KUKA KRL program: EPS_2_25716_MHLP03_A_20250903043914.src

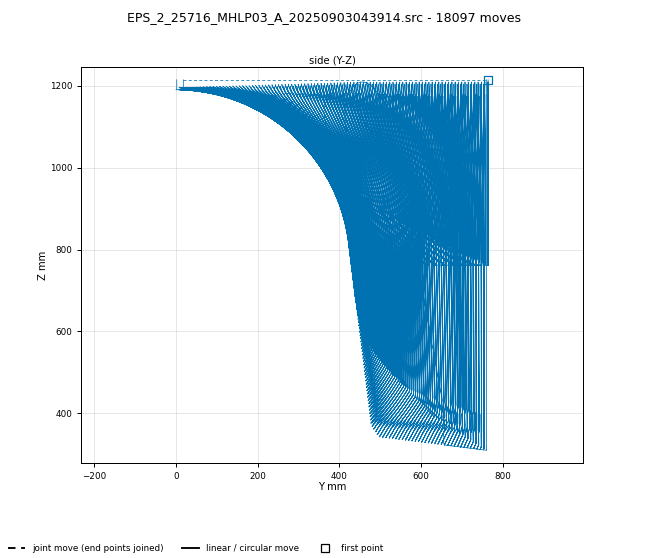
[picture p0: tool path of EPS_2_25716_MHLP03_A_20250903043914.src, 18097 of 18099 moves have a stored position in this frame; points joined in program order, loops and branches not executed]
&ACCESS RVP
&REL 4
&COMMENT QRS 19112012
&PARAM EDITMASK = *
DEF PART()
EXT BAS (BAS_COMMAND :IN,REAL :IN )
INT I
BAS (#INITMOV,0 )

;KUKA QRS Post kuka4.cps  Date:22-06-2017 !

File_ID=2811

QRS_PRE_INIT()

;Init var - Until changes are made in qrs_pre_init
Outlet_Square_prg=0
Inlet_1_Square_prg=0
Inlet_2_Square_prg=0
Inlet_3_Square_prg=0
Inlet_4_Square_prg=0
Inlet_5_Square_prg=0

Outlet_1={X 0.000, Y 457.000, Z 786.000, B 0.000, E1 0.000 }
Inlet_1={X 0.000, Y 514.000, Z 794.000, B 0.000, E1 180.000 }
Outlet_1_type=838
Inlet_1_type=762
;QRS#1=Sidecore dimensions
;QRS#2=825-33" Concrete
;QRS#3=750-30" Concrete
;QRS#4=
;QRS#5=
;QRS#6=
;QRS#7=
;QRS#8=
;QRS#9=S306-46
;QRS#10=S306-42L
;QRS#11=
;QRS#12=
;QRS#13=
;QRS#14=
;QRS#15=
;QRS#16=1524x152x1676 5,5'
;QRS#17=EPS Height
;QRS#18=1205
;QRS#19=*
;QRS#20= UPDATED VERSION 22-06-2017
;QRS#21=*
Outlet_Square=0650
Inlet_1_Square=0550
Inlet_2_Square=0
Inlet_3_Square=0
Inlet_4_Square=0
Inlet_5_Square=0
Mill_Square=1
Outlet_Square_Prg=267
Inlet_1_Square_prg=266

QRS_INIT()

$ADVANCE=5

; T1
PTP {E1 176.609,E2 176.609}
PTP {X 0,Y 763.422,A -85,B 0,C 180,E1 176.609,E2 176.609,E3 0,E4 0,E5 0,E6 0}
QRS_SPEED_INIT()
LIN {X 0,Y 763.422,Z 1215,A -85,B 0,C 180,E1 176.609,E2 176.609,E3 0,E4 0,E5 0,E6 0} C_VEL
LIN {X 0,Y 763.422,Z 764.06,A -85,B 0,C 180,E1 176.609,E2 176.609} C_VEL
LIN {X 0,Y 763.532,Z 762.06,A -85,B 0,C 180,E1 176.759,E2 176.759} C_VEL
LIN {X 0,Y 763.873,Z 762.06,A -85,B 0,C 180,E1 177.187,E2 177.187} C_VEL
LIN {X 0,Y 763.851,Z 762.06,A -85,B 0,C 180,E1 184.692,E2 184.692} C_VEL
LIN {X 0,Y 763.855,Z 762.06,A -85,B 0,C 180,E1 192.28,E2 192.28} C_VEL
LIN {X 0,Y 763.849,Z 762.06,A -85,B 0,C 180,E1 200.095,E2 200.095} C_VEL
LIN {X 0,Y 763.818,Z 762.06,A -85,B 0,C 180,E1 208.325,E2 208.325} C_VEL
LIN {X 0,Y 762.402,Z 762.06,A -85,B 0,C 180,E1 210.54,E2 210.54} C_VEL
LIN {X 0,Y 762.707,Z 762.06,A -85,B 0,C 180,E1 214.993,E2 214.993} C_VEL
LIN {X 0,Y 763.7,Z 762.06,A -85,B 0,C 180,E1 216.696,E2 216.696} C_VEL
LIN {X 0,Y 763.458,Z 762.06,A -85,B 0,C 180,E1 224.738,E2 224.738} C_VEL
LIN {X 0,Y 763.707,Z 762.06,A -85,B 0,C 180,E1 225.281,E2 225.281} C_VEL
LIN {X 0,Y 763.692,Z 762.06,A -85,B 0,C 180,E1 233.306,E2 233.306} C_VEL
LIN {X 0,Y 763.601,Z 762.06,A -85,B 0,C 180,E1 233.585,E2 233.585} C_VEL
LIN {X 0,Y 763.105,Z 765.194,A -85,B 0,C 180,E1 233.692,E2 233.692} C_VEL
LIN {X 0,Y 763.148,Z 825.436,A -85,B 0,C 180,E1 234.391,E2 234.391} C_VEL
LIN {X 0,Y 763.561,Z 841.683,A -85,B 0,C 180,E1 234.66,E2 234.66} C_VEL
LIN {X 0,Y 763.683,Z 859.427,A -85,B 0,C 180,E1 234.998,E2 234.998} C_VEL
LIN {X 0,Y 763.616,Z 876.824,A -85,B 0,C 180,E1 235.383,E2 235.383} C_VEL
LIN {X 0,Y 763.264,Z 892.857,A -85,B 0,C 180,E1 235.785,E2 235.785} C_VEL
LIN {X 0,Y 763.637,Z 914.318,A -85,B 0,C 180,E1 236.454,E2 236.454} C_VEL
LIN {X 0,Y 763.659,Z 936.004,A -85,B 0,C 180,E1 237.219,E2 237.219} C_VEL
LIN {X 0,Y 763.647,Z 955.467,A -85,B 0,C 180,E1 238,E2 238} C_VEL
LIN {X 0,Y 763.481,Z 968.047,A -85,B 0,C 180,E1 238.551,E2 238.551} C_VEL
LIN {X 0,Y 763.561,Z 976.645,A -85,B 0,C 180,E1 238.959,E2 238.959} C_VEL
LIN {X 0,Y 763.516,Z 991.062,A -85,B 0,C 180,E1 239.671,E2 239.671} C_VEL
LIN {X 0,Y 763.481,Z 1008.328,A -85,B 0,C 180,E1 240.608,E2 240.608} C_VEL
LIN {X 0,Y 763.638,Z 1024.577,A -85,B 0,C 180,E1 241.577,E2 241.577} C_VEL
LIN {X 0,Y 763.597,Z 1040.373,A -85,B 0,C 180,E1 242.594,E2 242.594} C_VEL
LIN {X 0,Y 763.3,Z 1055.415,A -85,B 0,C 180,E1 243.634,E2 243.634} C_VEL
LIN {X 0,Y 763.19,Z 1070.039,A -85,B 0,C 180,E1 244.738,E2 244.738} C_VEL
LIN {X 0,Y 763.448,Z 1083.461,A -85,B 0,C 180,E1 245.844,E2 245.844} C_VEL
LIN {X 0,Y 763.685,Z 1096.518,A -85,B 0,C 180,E1 247.003,E2 247.003} C_VEL
LIN {X 0,Y 763.163,Z 1110.025,A -85,B 0,C 180,E1 248.281,E2 248.281} C_VEL
LIN {X 0,Y 762.921,Z 1121.8,A -85,B 0,C 180,E1 249.497,E2 249.497} C_VEL
LIN {X 0,Y 763.255,Z 1133.583,A -85,B 0,C 180,E1 250.839,E2 250.839} C_VEL
LIN {X 0,Y 763.824,Z 1144.005,A -85,B 0,C 180,E1 252.135,E2 252.135} C_VEL
LIN {X 0,Y 763.053,Z 1154.834,A -85,B 0,C 180,E1 253.59,E2 253.59} C_VEL
LIN {X 0,Y 762.741,Z 1164.593,A -85,B 0,C 180,E1 255.058,E2 255.058} C_VEL
LIN {X 0,Y 763.114,Z 1172.36,A -85,B 0,C 180,E1 256.36,E2 256.36} C_VEL
LIN {X 0,Y 763.849,Z 1179.548,A -85,B 0,C 180,E1 257.72,E2 257.72} C_VEL
LIN {X 0,Y 762.886,Z 1187.414,A -85,B 0,C 180,E1 259.38,E2 259.38} C_VEL
LIN {X 0,Y 762.625,Z 1192.231,A -85,B 0,C 180,E1 260.568,E2 260.568} C_VEL
LIN {X 0,Y 762.79,Z 1195.675,A -85,B 0,C 180,E1 261.521,E2 261.521} C_VEL
LIN {X 0,Y 763.28,Z 1198.711,A -85,B 0,C 180,E1 262.474,E2 262.474} C_VEL
LIN {X 0,Y 763.858,Z 1201.343,A -85,B 0,C 180,E1 263.424,E2 263.424} C_VEL
LIN {X 0,Y 763.266,Z 1203.657,A -85,B 0,C 180,E1 264.362,E2 264.362} C_VEL
LIN {X 0,Y 762.79,Z 1205.612,A -85,B 0,C 180,E1 265.301,E2 265.301} C_VEL
LIN {X 0,Y 762.61,Z 1207.201,A -85,B 0,C 180,E1 266.242,E2 266.242} C_VEL
LIN {X 0,Y 762.976,Z 1208.861,A -85,B 0,C 180,E1 267.626,E2 267.626} C_VEL
LIN {X 0,Y 763.872,Z 1209.666,A -85,B 0,C 180,E1 269.062,E2 269.062} C_VEL
LIN {X 0,Y 762.824,Z 1209.715,A -85,B 0,C 180,E1 270.939,E2 270.939} C_VEL
LIN {X 0,Y 762.627,Z 1209.463,A -85,B 0,C 180,E1 271.621,E2 271.621} C_VEL
LIN {X 0,Y 762.799,Z 1208.402,A -85,B 0,C 180,E1 272.817,E2 272.817} C_VEL
LIN {X 0,Y 763.272,Z 1207.185,A -85,B 0,C 180,E1 273.755,E2 273.755} C_VEL
LIN {X 0,Y 763.867,Z 1205.576,A -85,B 0,C 180,E1 274.692,E2 274.692} C_VEL
LIN {X 0,Y 763.013,Z 1202.588,A -85,B 0,C 180,E1 276.111,E2 276.111} C_VEL
LIN {X 0,Y 762.637,Z 1198.716,A -85,B 0,C 180,E1 277.533,E2 277.533} C_VEL
LIN {X 0,Y 762.799,Z 1195.676,A -85,B 0,C 180,E1 278.479,E2 278.479} C_VEL
LIN {X 0,Y 763.569,Z 1190.398,A -85,B 0,C 180,E1 279.895,E2 279.895} C_VEL
LIN {X 0,Y 763.864,Z 1188.41,A -85,B 0,C 180,E1 280.367,E2 280.367} C_VEL
LIN {X 0,Y 763.206,Z 1182.983,A -85,B 0,C 180,E1 281.571,E2 281.571} C_VEL
LIN {X 0,Y 762.859,Z 1179.549,A -85,B 0,C 180,E1 282.296,E2 282.296} C_VEL
LIN {X 0,Y 762.736,Z 1172.081,A -85,B 0,C 180,E1 283.695,E2 283.695} C_VEL
LIN {X 0,Y 763.29,Z 1163.915,A -85,B 0,C 180,E1 285.044,E2 285.044} C_VEL
LIN {X 0,Y 763.763,Z 1158.34,A -85,B 0,C 180,E1 285.871,E2 285.871} C_VEL
LIN {X 0,Y 763.637,Z 1154.836,A -85,B 0,C 180,E1 286.397,E2 286.397} C_VEL
LIN {X 0,Y 762.912,Z 1144.007,A -85,B 0,C 180,E1 287.886,E2 287.886} C_VEL
LIN {X 0,Y 762.868,Z 1132,A -85,B 0,C 180,E1 289.358,E2 289.358} C_VEL
LIN {X 0,Y 763.42,Z 1120.423,A -85,B 0,C 180,E1 290.638,E2 290.638} C_VEL
LIN {X 0,Y 763.768,Z 1112.185,A -85,B 0,C 180,E1 291.477,E2 291.477} C_VEL
LIN {X 0,Y 763.558,Z 1105.856,A -85,B 0,C 180,E1 292.113,E2 292.113} C_VEL
LIN {X 0,Y 763.217,Z 1095.11,A -85,B 0,C 180,E1 293.14,E2 293.14} C_VEL
LIN {X 0,Y 763.154,Z 1081.968,A -85,B 0,C 180,E1 294.292,E2 294.292} C_VEL
LIN {X 0,Y 763.464,Z 1068.228,A -85,B 0,C 180,E1 295.394,E2 295.394} C_VEL
LIN {X 0,Y 763.662,Z 1053.606,A -85,B 0,C 180,E1 296.483,E2 296.483} C_VEL
LIN {X 0,Y 763.467,Z 1037.367,A -85,B 0,C 180,E1 297.609,E2 297.609} C_VEL
LIN {X 0,Y 763.402,Z 1021.787,A -85,B 0,C 180,E1 298.602,E2 298.602} C_VEL
LIN {X 0,Y 763.565,Z 1005.34,A -85,B 0,C 180,E1 299.557,E2 299.557} C_VEL
LIN {X 0,Y 763.602,Z 989.459,A -85,B 0,C 180,E1 300.411,E2 300.411} C_VEL
LIN {X 0,Y 763.621,Z 970.475,A -85,B 0,C 180,E1 301.335,E2 301.335} C_VEL
LIN {X 0,Y 763.591,Z 951.701,A -85,B 0,C 180,E1 302.16,E2 302.16} C_VEL
LIN {X 0,Y 763.574,Z 933.239,A -85,B 0,C 180,E1 302.888,E2 302.888} C_VEL
LIN {X 0,Y 763.35,Z 920.5,A -85,B 0,C 180,E1 303.348,E2 303.348} C_VEL
LIN {X 0,Y 763.571,Z 911.932,A -85,B 0,C 180,E1 303.623,E2 303.623} C_VEL
LIN {X 0,Y 763.721,Z 893.145,A -85,B 0,C 180,E1 304.183,E2 304.183} C_VEL
LIN {X 0,Y 763.708,Z 876.573,A -85,B 0,C 180,E1 304.618,E2 304.618} C_VEL
LIN {X 0,Y 763.517,Z 859.345,A -85,B 0,C 180,E1 305.013,E2 305.013} C_VEL
LIN {X 0,Y 763.205,Z 848.039,A -85,B 0,C 180,E1 305.249,E2 305.249} C_VEL
LIN {X 0,Y 763.489,Z 831.099,A -85,B 0,C 180,E1 305.51,E2 305.51} C_VEL
LIN {X 0,Y 763.501,Z 819.142,A -85,B 0,C 180,E1 305.669,E2 305.669} C_VEL
LIN {X 0,Y 763.102,Z 762.521,A -85,B 0,C 180,E1 306.339,E2 306.339} C_VEL
LIN {X 0,Y 763.722,Z 762.06,A -85,B 0,C 180,E1 306.444,E2 306.444} C_VEL
LIN {X 0,Y 763.585,Z 762.06,A -85,B 0,C 180,E1 306.961,E2 306.961} C_VEL
LIN {X 0,Y 763.809,Z 762.06,A -85,B 0,C 180,E1 312.129,E2 312.129} C_VEL
LIN {X 0,Y 763.614,Z 762.06,A -85,B 0,C 180,E1 312.57,E2 312.57} C_VEL
LIN {X 0,Y 763.761,Z 762.06,A -85,B 0,C 180,E1 320.266,E2 320.266} C_VEL
LIN {X 0,Y 763.673,Z 762.06,A -85,B 0,C 180,E1 326.571,E2 326.571} C_VEL
LIN {X 0,Y 763.435,Z 762.06,A -85,B 0,C 180,E1 327.303,E2 327.303} C_VEL
LIN {X 0,Y 763.817,Z 762.06,A -85,B 0,C 180,E1 333.784,E2 333.784} C_VEL
LIN {X 0,Y 763.847,Z 762.06,A -85,B 0,C 180,E1 341.889,E2 341.889} C_VEL
LIN {X 0,Y 763.863,Z 762.06,A -85,B 0,C 180,E1 349.632,E2 349.632} C_VEL
LIN {X 0,Y 763.842,Z 762.06,A -85,B 0,C 180,E1 357.187,E2 357.187} C_VEL
LIN {X 0,Y 763.858,Z 762.06,A -85,B 0,C 180,E1 364.692,E2 364.692} C_VEL
LIN {X 0,Y 763.826,Z 762.06,A -85,B 0,C 180,E1 372.28,E2 372.28} C_VEL
LIN {X 0,Y 763.82,Z 762.06,A -85,B 0,C 180,E1 380.096,E2 380.096} C_VEL
LIN {X 0,Y 763.775,Z 762.06,A -85,B 0,C 180,E1 388.327,E2 388.327} C_VEL
LIN {X 0,Y 763.769,Z 762.06,A -85,B 0,C 180,E1 394.938,E2 394.938} C_VEL
LIN {X 0,Y 762.467,Z 762.06,A -85,B 0,C 180,E1 399.734,E2 399.734} C_VEL
LIN {X 0,Y 763.757,Z 762.06,A -85,B 0,C 180,E1 402.134,E2 402.134} C_VEL
LIN {X 0,Y 763.589,Z 762.06,A -85,B 0,C 180,E1 402.569,E2 402.569} C_VEL
LIN {X 0,Y 763.857,Z 762.06,A -85,B 0,C 180,E1 410.259,E2 410.259} C_VEL
LIN {X 0,Y 763.738,Z 762.06,A -85,B 0,C 180,E1 416.565,E2 416.565} C_VEL
LIN {X 0,Y 763.397,Z 762.06,A -85,B 0,C 180,E1 416.915,E2 416.915} C_VEL
LIN {X 0,Y 762.602,Z 762.061,A -85,B 0,C 180,E1 416.991,E2 416.991} C_VEL
LIN {X 0,Y 763.35,Z 823.326,A -85,B 0,C 180,E1 417.706,E2 417.706} C_VEL
LIN {X 0,Y 763.333,Z 838.865,A -85,B 0,C 180,E1 417.911,E2 417.911} C_VEL
LIN {X 0,Y 763.673,Z 858.064,A -85,B 0,C 180,E1 418.263,E2 418.263} C_VEL
LIN {X 0,Y 763.723,Z 875.941,A -85,B 0,C 180,E1 418.651,E2 418.651} C_VEL
LIN {X 0,Y 763.595,Z 893.845,A -85,B 0,C 180,E1 419.106,E2 419.106} C_VEL
LIN {X 0,Y 763.455,Z 902.424,A -85,B 0,C 180,E1 419.354,E2 419.354} C_VEL
LIN {X 0,Y 763.674,Z 913.5,A -85,B 0,C 180,E1 419.706,E2 419.706} C_VEL
LIN {X 0,Y 763.678,Z 930.085,A -85,B 0,C 180,E1 420.28,E2 420.28} C_VEL
LIN {X 0,Y 763.697,Z 947.445,A -85,B 0,C 180,E1 420.959,E2 420.959} C_VEL
LIN {X 0,Y 763.678,Z 963.783,A -85,B 0,C 180,E1 421.67,E2 421.67} C_VEL
LIN {X 0,Y 763.609,Z 974.911,A -85,B 0,C 180,E1 422.198,E2 422.198} C_VEL
LIN {X 0,Y 763.613,Z 984.032,A -85,B 0,C 180,E1 422.661,E2 422.661} C_VEL
LIN {X 0,Y 763.513,Z 996.348,A -85,B 0,C 180,E1 423.315,E2 423.315} C_VEL
LIN {X 0,Y 763.537,Z 1011.273,A -85,B 0,C 180,E1 424.185,E2 424.185} C_VEL
LIN {X 0,Y 763.684,Z 1026.123,A -85,B 0,C 180,E1 425.134,E2 425.134} C_VEL
LIN {X 0,Y 763.619,Z 1038.484,A -85,B 0,C 180,E1 425.978,E2 425.978} C_VEL
LIN {X 0,Y 763.318,Z 1052.22,A -85,B 0,C 180,E1 426.991,E2 426.991} C_VEL
LIN {X 0,Y 763.258,Z 1064.783,A -85,B 0,C 180,E1 428.003,E2 428.003} C_VEL
LIN {X 0,Y 763.568,Z 1077.587,A -85,B 0,C 180,E1 429.134,E2 429.134} C_VEL
LIN {X 0,Y 763.744,Z 1087.004,A -85,B 0,C 180,E1 430.024,E2 430.024} C_VEL
LIN {X 0,Y 763.2,Z 1099.807,A -85,B 0,C 180,E1 431.321,E2 431.321} C_VEL
LIN {X 0,Y 763.019,Z 1110.232,A -85,B 0,C 180,E1 432.486,E2 432.486} C_VEL
LIN {X 0,Y 763.299,Z 1119.275,A -85,B 0,C 180,E1 433.595,E2 433.595} C_VEL
LIN {X 0,Y 763.838,Z 1128.649,A -85,B 0,C 180,E1 434.861,E2 434.861} C_VEL
LIN {X 0,Y 763.059,Z 1138.172,A -85,B 0,C 180,E1 436.263,E2 436.263} C_VEL
LIN {X 0,Y 762.712,Z 1144.936,A -85,B 0,C 180,E1 437.381,E2 437.381} C_VEL
LIN {X 0,Y 763.034,Z 1153.093,A -85,B 0,C 180,E1 438.905,E2 438.905} C_VEL
LIN {X 0,Y 763.728,Z 1158.659,A -85,B 0,C 180,E1 440.107,E2 440.107} C_VEL
LIN {X 0,Y 763.702,Z 1160.649,A -85,B 0,C 180,E1 440.582,E2 440.582} C_VEL
LIN {X 0,Y 763.147,Z 1164.462,A -85,B 0,C 180,E1 441.525,E2 441.525} C_VEL
LIN {X 0,Y 762.699,Z 1169.301,A -85,B 0,C 180,E1 442.941,E2 442.941} C_VEL
LIN {X 0,Y 763.043,Z 1173.205,A -85,B 0,C 180,E1 444.361,E2 444.361} C_VEL
LIN {X 0,Y 763.604,Z 1175.195,A -85,B 0,C 180,E1 445.306,E2 445.306} C_VEL
LIN {X 0,Y 763.572,Z 1176.903,A -85,B 0,C 180,E1 446.247,E2 446.247} C_VEL
LIN {X 0,Y 762.964,Z 1178.329,A -85,B 0,C 180,E1 447.184,E2 447.184} C_VEL
LIN {X 0,Y 762.58,Z 1179.53,A -85,B 0,C 180,E1 448.508,E2 448.508} C_VEL
LIN {X 0,Y 762.643,Z 1179.734,A -85,B 0,C 180,E1 449.061,E2 449.061} C_VEL
LIN {X 0,Y 763.561,Z 1179.673,A -85,B 0,C 180,E1 450.938,E2 450.938} C_VEL
LIN {X 0,Y 763.13,Z 1178.412,A -85,B 0,C 180,E1 452.638,E2 452.638} C_VEL
LIN {X 0,Y 762.743,Z 1176.796,A -85,B 0,C 180,E1 453.758,E2 453.758} C_VEL
LIN {X 0,Y 762.944,Z 1174.031,A -85,B 0,C 180,E1 455.169,E2 455.169} C_VEL
LIN {X 0,Y 763.153,Z 1172.957,A -85,B 0,C 180,E1 455.639,E2 455.639} C_VEL
LIN {X 0,Y 763.71,Z 1170.361,A -85,B 0,C 180,E1 456.577,E2 456.577} C_VEL
LIN {X 0,Y 763.728,Z 1168.983,A -85,B 0,C 180,E1 457.049,E2 457.049} C_VEL
LIN {X 0,Y 762.942,Z 1164.1,A -85,B 0,C 180,E1 458.477,E2 458.477} C_VEL
LIN {X 0,Y 762.689,Z 1159.333,A -85,B 0,C 180,E1 459.669,E2 459.669} C_VEL
LIN {X 0,Y 763.153,Z 1152.641,A -85,B 0,C 180,E1 461.094,E2 461.094} C_VEL
LIN {X 0,Y 763.854,Z 1146.251,A -85,B 0,C 180,E1 462.28,E2 462.28} C_VEL
LIN {X 0,Y 763.151,Z 1138.199,A -85,B 0,C 180,E1 463.641,E2 463.641} C_VEL
LIN {X 0,Y 762.78,Z 1128.325,A -85,B 0,C 180,E1 465.114,E2 465.114} C_VEL
LIN {X 0,Y 763.189,Z 1118.534,A -85,B 0,C 180,E1 466.407,E2 466.407} C_VEL
LIN {X 0,Y 763.808,Z 1108.38,A -85,B 0,C 180,E1 467.619,E2 467.619} C_VEL
LIN {X 0,Y 763.383,Z 1098.021,A -85,B 0,C 180,E1 468.775,E2 468.775} C_VEL
LIN {X 0,Y 763.102,Z 1086.005,A -85,B 0,C 180,E1 469.997,E2 469.997} C_VEL
LIN {X 0,Y 763.291,Z 1074.606,A -85,B 0,C 180,E1 471.054,E2 471.054} C_VEL
LIN {X 0,Y 763.698,Z 1062.183,A -85,B 0,C 180,E1 472.109,E2 472.109} C_VEL
LIN {X 0,Y 763.642,Z 1051.08,A -85,B 0,C 180,E1 472.999,E2 472.999} C_VEL
LIN {X 0,Y 763.363,Z 1037.208,A -85,B 0,C 180,E1 474.031,E2 474.031} C_VEL
LIN {X 0,Y 763.39,Z 1022.484,A -85,B 0,C 180,E1 475.026,E2 475.026} C_VEL
LIN {X 0,Y 763.608,Z 1007.982,A -85,B 0,C 180,E1 475.922,E2 475.922} C_VEL
LIN {X 0,Y 763.681,Z 992.341,A -85,B 0,C 180,E1 476.81,E2 476.81} C_VEL
LIN {X 0,Y 763.637,Z 977.185,A -85,B 0,C 180,E1 477.602,E2 477.602} C_VEL
LIN {X 0,Y 763.612,Z 960.801,A -85,B 0,C 180,E1 478.379,E2 478.379} C_VEL
LIN {X 0,Y 763.629,Z 942.917,A -85,B 0,C 180,E1 479.138,E2 479.138} C_VEL
LIN {X 0,Y 763.481,Z 932.728,A -85,B 0,C 180,E1 479.536,E2 479.536} C_VEL
LIN {X 0,Y 763.665,Z 923.871,A -85,B 0,C 180,E1 479.851,E2 479.851} C_VEL
LIN {X 0,Y 763.752,Z 908.211,A -85,B 0,C 180,E1 480.371,E2 480.371} C_VEL
LIN {X 0,Y 763.742,Z 891.43,A -85,B 0,C 180,E1 480.865,E2 480.865} C_VEL
LIN {X 0,Y 763.585,Z 872.972,A -85,B 0,C 180,E1 481.335,E2 481.335} C_VEL
LIN {X 0,Y 763.349,Z 865.666,A -85,B 0,C 180,E1 481.501,E2 481.501} C_VEL
LIN {X 0,Y 763.643,Z 854.355,A -85,B 0,C 180,E1 481.72,E2 481.72} C_VEL
LIN {X 0,Y 763.767,Z 835.648,A -85,B 0,C 180,E1 482.025,E2 482.025} C_VEL
LIN {X 0,Y 763.645,Z 814.716,A -85,B 0,C 180,E1 482.292,E2 482.292} C_VEL
LIN {X 0,Y 763.119,Z 784.369,A -85,B 0,C 180,E1 482.649,E2 482.649} C_VEL
LIN {X 0,Y 761.841,Z 762.933,A -85,B 0,C 180,E1 482.946,E2 482.946} C_VEL
LIN {X 0,Y 761.836,Z 762.06,A -85,B 0,C 180,E1 482.963,E2 482.963} C_VEL
LIN {X 0,Y 762.124,Z 762.06,A -85,B 0,C 180,E1 482.976,E2 482.976} C_VEL
LIN {X 0,Y 763.606,Z 762.06,A -85,B 0,C 180,E1 483.119,E2 483.119} C_VEL
LIN {X 0,Y 763.812,Z 762.06,A -85,B 0,C 180,E1 483.443,E2 483.443} C_VEL
LIN {X 0,Y 763.69,Z 762.06,A -85,B 0,C 180,E1 486.694,E2 486.694} C_VEL
LIN {X 0,Y 763.69,Z 762.06,A -85,B 0,C 180,E1 494.72,E2 494.72} C_VEL
LIN {X 0,Y 763.483,Z 762.06,A -85,B 0,C 180,E1 495.264,E2 495.264} C_VEL
LIN {X 0,Y 762.408,Z 762.06,A -85,B 0,C 180,E1 500.389,E2 500.389} C_VEL
LIN {X 0,Y 763.783,Z 762.06,A -85,B 0,C 180,E1 502.743,E2 502.743} C_VEL
LIN {X 0,Y 763.683,Z 762.06,A -85,B 0,C 180,E1 510.145,E2 510.145} C_VEL
LIN {X 0,Y 762.968,Z 762.06,A -85,B 0,C 180,E1 511.64,E2 511.64} C_VEL
LIN {X 0,Y 763.8,Z 762.06,A -85,B 0,C 180,E1 517.894,E2 517.894} C_VEL
LIN {X 0,Y 763.495,Z 762.06,A -85,B 0,C 180,E1 524.953,E2 524.953} C_VEL
LIN {X 0,Y 763.693,Z 762.06,A -85,B 0,C 180,E1 525.791,E2 525.791} C_VEL
LIN {X 0,Y 763.845,Z 762.06,A -85,B 0,C 180,E1 529.632,E2 529.632} C_VEL
LIN {X 0,Y 763.532,Z 762.06,A -85,B 0,C 180,E1 536.759,E2 536.759} C_VEL
LIN {X 0,Y 754.518,Z 762.06,A -85,B 0,C 180,E1 539.358,E2 539.358} C_VEL
LIN {X 0,Y 754.715,Z 762.06,A -85,B 0,C 180,E1 546.362,E2 546.362} C_VEL
LIN {X 0,Y 755.003,Z 762.06,A -85,B 0,C 180,E1 553.379,E2 553.379} C_VEL
LIN {X 0,Y 755.112,Z 762.06,A -85,B 0,C 180,E1 560.95,E2 560.95} C_VEL
LIN {X 0,Y 754.911,Z 762.06,A -85,B 0,C 180,E1 569.525,E2 569.525} C_VEL
LIN {X 0,Y 754.735,Z 762.06,A -85,B 0,C 180,E1 577.848,E2 577.848} C_VEL
LIN {X 0,Y 754.995,Z 762.06,A -85,B 0,C 180,E1 586.132,E2 586.132} C_VEL
LIN {X 0,Y 755.889,Z 764.005,A -85,B 0,C 180,E1 593.275,E2 593.275} C_VEL
LIN {X 0,Y 757.067,Z 866.417,A -85,B 0,C 180,E1 594.797,E2 594.797} C_VEL
LIN {X 0,Y 756.732,Z 937.533,A -85,B 0,C 180,E1 596.942,E2 596.942} C_VEL
LIN {X 0,Y 756.224,Z 1008.772,A -85,B 0,C 180,E1 600.324,E2 600.324} C_VEL
LIN {X 0,Y 755.596,Z 1073.515,A -85,B 0,C 180,E1 604.753,E2 604.753} C_VEL
LIN {X 0,Y 755.135,Z 1125.789,A -85,B 0,C 180,E1 609.73,E2 609.73} C_VEL
LIN {X 0,Y 754.862,Z 1162.477,A -85,B 0,C 180,E1 614.561,E2 614.561} C_VEL
LIN {X 0,Y 754.828,Z 1188.719,A -85,B 0,C 180,E1 619.581,E2 619.581} C_VEL
LIN {X 0,Y 755.026,Z 1204.76,A -85,B 0,C 180,E1 624.813,E2 624.813} C_VEL
LIN {X 0,Y 755.621,Z 1209.837,A -85,B 0,C 180,E1 629.424,E2 629.424} C_VEL
LIN {X 0,Y 755.519,Z 1204.764,A -85,B 0,C 180,E1 635.181,E2 635.181} C_VEL
LIN {X 0,Y 755.373,Z 1184.858,A -85,B 0,C 180,E1 641.287,E2 641.287} C_VEL
LIN {X 0,Y 755.345,Z 1150.798,A -85,B 0,C 180,E1 647.144,E2 647.144} C_VEL
LIN {X 0,Y 755.668,Z 1103.645,A -85,B 0,C 180,E1 652.569,E2 652.569} C_VEL
LIN {X 0,Y 756.059,Z 1043.633,A -85,B 0,C 180,E1 657.472,E2 657.472} C_VEL
LIN {X 0,Y 756.496,Z 976.301,A -85,B 0,C 180,E1 661.381,E2 661.381} C_VEL
LIN {X 0,Y 756.901,Z 903.888,A -85,B 0,C 180,E1 664.21,E2 664.21} C_VEL
LIN {X 0,Y 756.982,Z 829.369,A -85,B 0,C 180,E1 665.888,E2 665.888} C_VEL
LIN {X 0,Y 755.632,Z 762.06,A -85,B 0,C 180,E1 666.796,E2 666.796} C_VEL
LIN {X 0,Y 754.653,Z 762.06,A -85,B 0,C 180,E1 673.89,E2 673.89} C_VEL
LIN {X 0,Y 754.78,Z 762.06,A -85,B 0,C 180,E1 682.154,E2 682.154} C_VEL
LIN {X 0,Y 754.74,Z 762.06,A -85,B 0,C 180,E1 688.643,E2 688.643} C_VEL
LIN {X 0,Y 755.303,Z 762.06,A -85,B 0,C 180,E1 694.389,E2 694.389} C_VEL
LIN {X 0,Y 754.964,Z 762.06,A -85,B 0,C 180,E1 703.039,E2 703.039} C_VEL
LIN {X 0,Y 755.425,Z 762.06,A -85,B 0,C 180,E1 710.155,E2 710.155} C_VEL
LIN {X 0,Y 755.038,Z 762.06,A -85,B 0,C 180,E1 718.26,E2 718.26} C_VEL
LIN {X 0,Y 754.869,Z 762.06,A -85,B 0,C 180,E1 726.055,E2 726.055} C_VEL
LIN {X 0,Y 754.978,Z 762.06,A -85,B 0,C 180,E1 733.355,E2 733.355} C_VEL
LIN {X 0,Y 755.074,Z 762.06,A -85,B 0,C 180,E1 740.949,E2 740.949} C_VEL
LIN {X 0,Y 755.031,Z 762.06,A -85,B 0,C 180,E1 749.492,E2 749.492} C_VEL
LIN {X 0,Y 754.827,Z 762.06,A -85,B 0,C 180,E1 756.369,E2 756.369} C_VEL
LIN {X 0,Y 755.347,Z 762.06,A -85,B 0,C 180,E1 762.879,E2 762.879} C_VEL
LIN {X 0,Y 755.489,Z 762.06,A -85,B 0,C 180,E1 770.781,E2 770.781} C_VEL
LIN {X 0,Y 755.761,Z 763.481,A -85,B 0,C 180,E1 776.67,E2 776.67} C_VEL
LIN {X 0,Y 756.835,Z 867.232,A -85,B 0,C 180,E1 778.14,E2 778.14} C_VEL
LIN {X 0,Y 756.556,Z 937.416,A -85,B 0,C 180,E1 780.258,E2 780.258} C_VEL
LIN {X 0,Y 756.087,Z 1005.684,A -85,B 0,C 180,E1 783.576,E2 783.576} C_VEL
LIN {X 0,Y 755.561,Z 1064.464,A -85,B 0,C 180,E1 787.739,E2 787.739} C_VEL
LIN {X 0,Y 755.151,Z 1110.654,A -85,B 0,C 180,E1 792.35,E2 792.35} C_VEL
LIN {X 0,Y 754.843,Z 1143.269,A -85,B 0,C 180,E1 796.968,E2 796.968} C_VEL
LIN {X 0,Y 754.988,Z 1166.131,A -85,B 0,C 180,E1 801.918,E2 801.918} C_VEL
LIN {X 0,Y 755.023,Z 1178.299,A -85,B 0,C 180,E1 807.123,E2 807.123} C_VEL
LIN {X 0,Y 755.288,Z 1179.26,A -85,B 0,C 180,E1 811.727,E2 811.727} C_VEL
LIN {X 0,Y 755.439,Z 1167.758,A -85,B 0,C 180,E1 817.499,E2 817.499} C_VEL
LIN {X 0,Y 755.48,Z 1142.577,A -85,B 0,C 180,E1 823.047,E2 823.047} C_VEL
LIN {X 0,Y 755.644,Z 1102.95,A -85,B 0,C 180,E1 828.428,E2 828.428} C_VEL
LIN {X 0,Y 755.962,Z 1050.543,A -85,B 0,C 180,E1 833.287,E2 833.287} C_VEL
LIN {X 0,Y 756.297,Z 988.391,A -85,B 0,C 180,E1 837.304,E2 837.304} C_VEL
LIN {X 0,Y 756.657,Z 919.117,A -85,B 0,C 180,E1 840.32,E2 840.32} C_VEL
LIN {X 0,Y 756.897,Z 847.457,A -85,B 0,C 180,E1 842.156,E2 842.156} C_VEL
LIN {X 0,Y 755.541,Z 762.06,A -85,B 0,C 180,E1 843.332,E2 843.332} C_VEL
LIN {X 0,Y 754.065,Z 762.06,A -85,B 0,C 180,E1 849.31,E2 849.31} C_VEL
LIN {X 0,Y 754.889,Z 762.06,A -85,B 0,C 180,E1 856.095,E2 856.095} C_VEL
LIN {X 0,Y 755.09,Z 762.06,A -85,B 0,C 180,E1 863.646,E2 863.646} C_VEL
LIN {X 0,Y 754.879,Z 762.06,A -85,B 0,C 180,E1 871.816,E2 871.816} C_VEL
LIN {X 0,Y 754.77,Z 762.06,A -85,B 0,C 180,E1 879.408,E2 879.408} C_VEL
LIN {X 0,Y 755.411,Z 762.06,A -85,B 0,C 180,E1 886.824,E2 886.824} C_VEL
LIN {X 0,Y 754.221,Z 762.06,A -85,B 0,C 180,E1 893.657,E2 893.657} C_VEL
LIN {X 0,Y 755.069,Z 762.06,A -85,B 0,C 180,E1 898.284,E2 898.284} C_VEL
LIN {X 0,Y 754.518,Z 762.06,A -85,B 0,C 180,E1 899.358,E2 899.358} C_VEL
LIN {X 0,Y 746.381,Z 762.06,A -85,B 0,C 180,E1 901.989,E2 901.989} C_VEL
LIN {X 0,Y 746.269,Z 762.06,A -85,B 0,C 180,E1 907.609,E2 907.609} C_VEL
LIN {X 0,Y 746.903,Z 762.06,A -85,B 0,C 180,E1 913.527,E2 913.527} C_VEL
LIN {X 0,Y 747.198,Z 762.06,A -85,B 0,C 180,E1 920.836,E2 920.836} C_VEL
LIN {X 0,Y 747.486,Z 762.06,A -85,B 0,C 180,E1 928.515,E2 928.515} C_VEL
LIN {X 0,Y 747.242,Z 762.06,A -85,B 0,C 180,E1 936.828,E2 936.828} C_VEL
LIN {X 0,Y 746.946,Z 762.06,A -85,B 0,C 180,E1 946.184,E2 946.184} C_VEL
LIN {X 0,Y 747.356,Z 763.412,A -85,B 0,C 180,E1 952.778,E2 952.778} C_VEL
LIN {X 0,Y 750.226,Z 775.649,A -85,B 0,C 180,E1 953.088,E2 953.088} C_VEL
LIN {X 0,Y 750.485,Z 865.241,A -85,B 0,C 180,E1 954.415,E2 954.415} C_VEL
LIN {X 0,Y 749.898,Z 935.677,A -85,B 0,C 180,E1 956.526,E2 956.526} C_VEL
LIN {X 0,Y 749.014,Z 1006.369,A -85,B 0,C 180,E1 959.866,E2 959.866} C_VEL
LIN {X 0,Y 748.042,Z 1071.316,A -85,B 0,C 180,E1 964.296,E2 964.296} C_VEL
LIN {X 0,Y 747.318,Z 1123.096,A -85,B 0,C 180,E1 969.198,E2 969.198} C_VEL
LIN {X 0,Y 747.022,Z 1160.497,A -85,B 0,C 180,E1 974.093,E2 974.093} C_VEL
LIN {X 0,Y 747,Z 1187.51,A -85,B 0,C 180,E1 979.175,E2 979.175} C_VEL
LIN {X 0,Y 747.062,Z 1204.76,A -85,B 0,C 180,E1 984.758,E2 984.758} C_VEL
LIN {X 0,Y 747.615,Z 1209.837,A -85,B 0,C 180,E1 989.418,E2 989.418} C_VEL
LIN {X 0,Y 747.495,Z 1204.764,A -85,B 0,C 180,E1 995.237,E2 995.237} C_VEL
LIN {X 0,Y 747.349,Z 1184.859,A -85,B 0,C 180,E1 1001.41,E2 1001.41} C_VEL
LIN {X 0,Y 747.385,Z 1151.064,A -85,B 0,C 180,E1 1007.296,E2 1007.296} C_VEL
LIN {X 0,Y 747.909,Z 1103.128,A -85,B 0,C 180,E1 1012.866,E2 1012.866} C_VEL
LIN {X 0,Y 748.596,Z 1043.549,A -85,B 0,C 180,E1 1017.776,E2 1017.776} C_VEL
LIN {X 0,Y 749.437,Z 974.405,A -85,B 0,C 180,E1 1021.807,E2 1021.807} C_VEL
LIN {X 0,Y 750.191,Z 902.761,A -85,B 0,C 180,E1 1024.595,E2 1024.595} C_VEL
LIN {X 0,Y 750.507,Z 828.895,A -85,B 0,C 180,E1 1026.253,E2 1026.253} C_VEL
LIN {X 0,Y 748.657,Z 766.226,A -85,B 0,C 180,E1 1027.113,E2 1027.113} C_VEL
LIN {X 0,Y 747.392,Z 762.06,A -85,B 0,C 180,E1 1027.323,E2 1027.323} C_VEL
LIN {X 0,Y 746.72,Z 762.06,A -85,B 0,C 180,E1 1033.797,E2 1033.797} C_VEL
LIN {X 0,Y 746.941,Z 762.06,A -85,B 0,C 180,E1 1041.686,E2 1041.686} C_VEL
LIN {X 0,Y 746.71,Z 762.06,A -85,B 0,C 180,E1 1048.766,E2 1048.766} C_VEL
LIN {X 0,Y 746.635,Z 762.06,A -85,B 0,C 180,E1 1055.358,E2 1055.358} C_VEL
LIN {X 0,Y 747.083,Z 762.06,A -85,B 0,C 180,E1 1062.855,E2 1062.855} C_VEL
LIN {X 0,Y 746.761,Z 762.06,A -85,B 0,C 180,E1 1071.22,E2 1071.22} C_VEL
LIN {X 0,Y 747.042,Z 762.06,A -85,B 0,C 180,E1 1078.242,E2 1078.242} C_VEL
LIN {X 0,Y 747.42,Z 762.06,A -85,B 0,C 180,E1 1085.231,E2 1085.231} C_VEL
LIN {X 0,Y 746.878,Z 762.06,A -85,B 0,C 180,E1 1093.503,E2 1093.503} C_VEL
LIN {X 0,Y 747.177,Z 762.06,A -85,B 0,C 180,E1 1100.811,E2 1100.811} C_VEL
LIN {X 0,Y 747.487,Z 762.06,A -85,B 0,C 180,E1 1108.488,E2 1108.488} C_VEL
LIN {X 0,Y 747.423,Z 762.06,A -85,B 0,C 180,E1 1115.348,E2 1115.348} C_VEL
LIN {X 0,Y 747.352,Z 762.06,A -85,B 0,C 180,E1 1122.855,E2 1122.855} C_VEL
LIN {X 0,Y 747.012,Z 762.06,A -85,B 0,C 180,E1 1131.745,E2 1131.745} C_VEL
LIN {X 0,Y 747.693,Z 763.504,A -85,B 0,C 180,E1 1136.263,E2 1136.263} C_VEL
LIN {X 0,Y 749.982,Z 870.345,A -85,B 0,C 180,E1 1137.882,E2 1137.882} C_VEL
LIN {X 0,Y 749.446,Z 940.007,A -85,B 0,C 180,E1 1140.05,E2 1140.05} C_VEL
LIN {X 0,Y 748.647,Z 1007.499,A -85,B 0,C 180,E1 1143.4,E2 1143.4} C_VEL
LIN {X 0,Y 747.828,Z 1066.541,A -85,B 0,C 180,E1 1147.682,E2 1147.682} C_VEL
LIN {X 0,Y 747.273,Z 1113.087,A -85,B 0,C 180,E1 1152.462,E2 1152.462} C_VEL
LIN {X 0,Y 746.848,Z 1144.559,A -85,B 0,C 180,E1 1157.045,E2 1157.045} C_VEL
LIN {X 0,Y 747.023,Z 1166.13,A -85,B 0,C 180,E1 1161.831,E2 1161.831} C_VEL
LIN {X 0,Y 747.044,Z 1178.299,A -85,B 0,C 180,E1 1167.092,E2 1167.092} C_VEL
LIN {X 0,Y 747.28,Z 1179.261,A -85,B 0,C 180,E1 1171.746,E2 1171.746} C_VEL
LIN {X 0,Y 747.394,Z 1167.76,A -85,B 0,C 180,E1 1177.58,E2 1177.58} C_VEL
LIN {X 0,Y 747.405,Z 1141.98,A -85,B 0,C 180,E1 1183.292,E2 1183.292} C_VEL
LIN {X 0,Y 747.739,Z 1102.471,A -85,B 0,C 180,E1 1188.685,E2 1188.685} C_VEL
LIN {X 0,Y 748.26,Z 1049.836,A -85,B 0,C 180,E1 1193.595,E2 1193.595} C_VEL
LIN {X 0,Y 748.976,Z 987.217,A -85,B 0,C 180,E1 1197.657,E2 1197.657} C_VEL
LIN {X 0,Y 749.656,Z 917.982,A -85,B 0,C 180,E1 1200.674,E2 1200.674} C_VEL
LIN {X 0,Y 750.131,Z 846.617,A -85,B 0,C 180,E1 1202.497,E2 1202.497} C_VEL
LIN {X 0,Y 747.7,Z 762.06,A -85,B 0,C 180,E1 1203.766,E2 1203.766} C_VEL
LIN {X 0,Y 745.884,Z 762.06,A -85,B 0,C 180,E1 1211.361,E2 1211.361} C_VEL
LIN {X 0,Y 746.865,Z 762.06,A -85,B 0,C 180,E1 1216.125,E2 1216.125} C_VEL
LIN {X 0,Y 747.206,Z 762.06,A -85,B 0,C 180,E1 1223.293,E2 1223.293} C_VEL
LIN {X 0,Y 746.765,Z 762.06,A -85,B 0,C 180,E1 1232.056,E2 1232.056} C_VEL
LIN {X 0,Y 746.917,Z 762.06,A -85,B 0,C 180,E1 1239.182,E2 1239.182} C_VEL
LIN {X 0,Y 747.371,Z 762.06,A -85,B 0,C 180,E1 1247.7,E2 1247.7} C_VEL
LIN {X 0,Y 747.793,Z 762.06,A -85,B 0,C 180,E1 1257.103,E2 1257.103} C_VEL
LIN {X 0,Y 746.381,Z 762.06,A -85,B 0,C 180,E1 1261.989,E2 1261.989} C_VEL
LIN {X 0,Y 739.308,Z 762.06,A -85,B 0,C 180,E1 1264.67,E2 1264.67} C_VEL
LIN {X 0,Y 738.81,Z 762.06,A -85,B 0,C 180,E1 1273.678,E2 1273.678} C_VEL
LIN {X 0,Y 739.005,Z 762.06,A -85,B 0,C 180,E1 1281.078,E2 1281.078} C_VEL
LIN {X 0,Y 738.995,Z 762.06,A -85,B 0,C 180,E1 1289.288,E2 1289.288} C_VEL
LIN {X 0,Y 738.669,Z 762.06,A -85,B 0,C 180,E1 1297.774,E2 1297.774} C_VEL
LIN {X 0,Y 738.696,Z 762.06,A -85,B 0,C 180,E1 1306.547,E2 1306.547} C_VEL
LIN {X 0,Y 738.943,Z 763.295,A -85,B 0,C 180,E1 1312.28,E2 1312.28} C_VEL
LIN {X 0,Y 743.829,Z 774.833,A -85,B 0,C 180,E1 1312.708,E2 1312.708} C_VEL
LIN {X 0,Y 743.911,Z 865.753,A -85,B 0,C 180,E1 1314.064,E2 1314.064} C_VEL
LIN {X 0,Y 743.056,Z 936.392,A -85,B 0,C 180,E1 1316.206,E2 1316.206} C_VEL
LIN {X 0,Y 741.79,Z 1007.864,A -85,B 0,C 180,E1 1319.632,E2 1319.632} C_VEL
LIN {X 0,Y 740.447,Z 1072.965,A -85,B 0,C 180,E1 1324.153,E2 1324.153} C_VEL
LIN {X 0,Y 739.475,Z 1124.923,A -85,B 0,C 180,E1 1329.18,E2 1329.18} C_VEL
LIN {X 0,Y 739.077,Z 1161.839,A -85,B 0,C 180,E1 1334.124,E2 1334.124} C_VEL
LIN {X 0,Y 738.961,Z 1188.72,A -85,B 0,C 180,E1 1339.355,E2 1339.355} C_VEL
LIN {X 0,Y 739.097,Z 1204.76,A -85,B 0,C 180,E1 1344.701,E2 1344.701} C_VEL
LIN {X 0,Y 738.97,Z 1209.838,A -85,B 0,C 180,E1 1350.587,E2 1350.587} C_VEL
LIN {X 0,Y 739.156,Z 1203.527,A -85,B 0,C 180,E1 1355.886,E2 1355.886} C_VEL
LIN {X 0,Y 739.187,Z 1183.504,A -85,B 0,C 180,E1 1361.838,E2 1361.838} C_VEL
LIN {X 0,Y 739.379,Z 1150.632,A -85,B 0,C 180,E1 1367.55,E2 1367.55} C_VEL
LIN {X 0,Y 740.182,Z 1104.396,A -85,B 0,C 180,E1 1372.994,E2 1372.994} C_VEL
LIN {X 0,Y 741.152,Z 1044.098,A -85,B 0,C 180,E1 1378.039,E2 1378.039} C_VEL
LIN {X 0,Y 742.395,Z 974.979,A -85,B 0,C 180,E1 1382.115,E2 1382.115} C_VEL
LIN {X 0,Y 743.495,Z 902.383,A -85,B 0,C 180,E1 1384.964,E2 1384.964} C_VEL
LIN {X 0,Y 744.055,Z 829.493,A -85,B 0,C 180,E1 1386.609,E2 1386.609} C_VEL
LIN {X 0,Y 742.194,Z 768.894,A -85,B 0,C 180,E1 1387.459,E2 1387.459} C_VEL
LIN {X 0,Y 739.235,Z 762.06,A -85,B 0,C 180,E1 1387.75,E2 1387.75} C_VEL
LIN {X 0,Y 738.941,Z 762.06,A -85,B 0,C 180,E1 1393.432,E2 1393.432} C_VEL
LIN {X 0,Y 739.092,Z 762.06,A -85,B 0,C 180,E1 1401.203,E2 1401.203} C_VEL
LIN {X 0,Y 738.816,Z 762.06,A -85,B 0,C 180,E1 1408.41,E2 1408.41} C_VEL
LIN {X 0,Y 738.809,Z 762.06,A -85,B 0,C 180,E1 1415.079,E2 1415.079} C_VEL
LIN {X 0,Y 739.142,Z 762.06,A -85,B 0,C 180,E1 1422.665,E2 1422.665} C_VEL
LIN {X 0,Y 738.811,Z 762.06,A -85,B 0,C 180,E1 1431.124,E2 1431.124} C_VEL
LIN {X 0,Y 739.045,Z 762.06,A -85,B 0,C 180,E1 1438.223,E2 1438.223} C_VEL
LIN {X 0,Y 739.111,Z 762.06,A -85,B 0,C 180,E1 1445.672,E2 1445.672} C_VEL
LIN {X 0,Y 738.812,Z 762.06,A -85,B 0,C 180,E1 1453.653,E2 1453.653} C_VEL
LIN {X 0,Y 739.011,Z 762.06,A -85,B 0,C 180,E1 1461.052,E2 1461.052} C_VEL
LIN {X 0,Y 739.079,Z 762.06,A -85,B 0,C 180,E1 1469.304,E2 1469.304} C_VEL
LIN {X 0,Y 739.091,Z 762.06,A -85,B 0,C 180,E1 1475.859,E2 1475.859} C_VEL
LIN {X 0,Y 738.917,Z 762.06,A -85,B 0,C 180,E1 1483.465,E2 1483.465} C_VEL
LIN {X 0,Y 739.163,Z 762.06,A -85,B 0,C 180,E1 1491.264,E2 1491.264} C_VEL
LIN {X 0,Y 739.538,Z 764.008,A -85,B 0,C 180,E1 1495.847,E2 1495.847} C_VEL
LIN {X 0,Y 742.658,Z 776.73,A -85,B 0,C 180,E1 1496.155,E2 1496.155} C_VEL
LIN {X 0,Y 743.156,Z 868.937,A -85,B 0,C 180,E1 1497.52,E2 1497.52} C_VEL
LIN {X 0,Y 742.369,Z 939.044,A -85,B 0,C 180,E1 1499.696,E2 1499.696} C_VEL
LIN {X 0,Y 741.255,Z 1007.212,A -85,B 0,C 180,E1 1503.097,E2 1503.097} C_VEL
LIN {X 0,Y 740.13,Z 1067.214,A -85,B 0,C 180,E1 1507.498,E2 1507.498} C_VEL
LIN {X 0,Y 739.39,Z 1114.521,A -85,B 0,C 180,E1 1512.45,E2 1512.45} C_VEL
LIN {X 0,Y 738.854,Z 1146.779,A -85,B 0,C 180,E1 1517.308,E2 1517.308} C_VEL
LIN {X 0,Y 739.064,Z 1166.128,A -85,B 0,C 180,E1 1521.743,E2 1521.743} C_VEL
LIN {X 0,Y 739.053,Z 1178.298,A -85,B 0,C 180,E1 1527.061,E2 1527.061} C_VEL
LIN {X 0,Y 739.272,Z 1179.261,A -85,B 0,C 180,E1 1531.764,E2 1531.764} C_VEL
LIN {X 0,Y 739.373,Z 1167.762,A -85,B 0,C 180,E1 1537.663,E2 1537.663} C_VEL
LIN {X 0,Y 739.384,Z 1141.932,A -85,B 0,C 180,E1 1543.448,E2 1543.448} C_VEL
LIN {X 0,Y 739.846,Z 1101.867,A -85,B 0,C 180,E1 1548.962,E2 1548.962} C_VEL
LIN {X 0,Y 740.623,Z 1049.447,A -85,B 0,C 180,E1 1553.884,E2 1553.884} C_VEL
LIN {X 0,Y 741.63,Z 986.72,A -85,B 0,C 180,E1 1557.983,E2 1557.983} C_VEL
LIN {X 0,Y 742.691,Z 917.302,A -85,B 0,C 180,E1 1561.018,E2 1561.018} C_VEL
LIN {X 0,Y 743.351,Z 847.414,A -85,B 0,C 180,E1 1562.817,E2 1562.817} C_VEL
LIN {X 0,Y 740.57,Z 765.741,A -85,B 0,C 180,E1 1563.989,E2 1563.989} C_VEL
LIN {X 0,Y 739.58,Z 762.06,A -85,B 0,C 180,E1 1564.327,E2 1564.327} C_VEL
LIN {X 0,Y 738.7,Z 762.06,A -85,B 0,C 180,E1 1573.453,E2 1573.453} C_VEL
LIN {X 0,Y 739.104,Z 762.06,A -85,B 0,C 180,E1 1582.728,E2 1582.728} C_VEL
LIN {X 0,Y 739.028,Z 762.06,A -85,B 0,C 180,E1 1591.156,E2 1591.156} C_VEL
LIN {X 0,Y 738.968,Z 762.06,A -85,B 0,C 180,E1 1599.031,E2 1599.031} C_VEL
LIN {X 0,Y 739.365,Z 762.06,A -85,B 0,C 180,E1 1607.565,E2 1607.565} C_VEL
LIN {X 0,Y 739.752,Z 762.06,A -85,B 0,C 180,E1 1617.072,E2 1617.072} C_VEL
LIN {X 0,Y 739.308,Z 762.06,A -85,B 0,C 180,E1 1624.67,E2 1624.67} C_VEL
LIN {X 0,Y 730.335,Z 762.06,A -85,B 0,C 180,E1 1627.348,E2 1627.348} C_VEL
LIN {X 0,Y 730.723,Z 762.06,A -85,B 0,C 180,E1 1633.832,E2 1633.832} C_VEL
LIN {X 0,Y 730.832,Z 762.06,A -85,B 0,C 180,E1 1641.325,E2 1641.325} C_VEL
LIN {X 0,Y 731.041,Z 762.06,A -85,B 0,C 180,E1 1649.217,E2 1649.217} C_VEL
LIN {X 0,Y 730.651,Z 762.06,A -85,B 0,C 180,E1 1657.809,E2 1657.809} C_VEL
LIN {X 0,Y 730.884,Z 762.06,A -85,B 0,C 180,E1 1665.964,E2 1665.964} C_VEL
LIN {X 0,Y 730.807,Z 764.041,A -85,B 0,C 180,E1 1671.794,E2 1671.794} C_VEL
LIN {X 0,Y 737.481,Z 777.622,A -85,B 0,C 180,E1 1672.365,E2 1672.365} C_VEL
LIN {X 0,Y 737.366,Z 867.033,A -85,B 0,C 180,E1 1673.725,E2 1673.725} C_VEL
LIN {X 0,Y 736.196,Z 937.434,A -85,B 0,C 180,E1 1675.891,E2 1675.891} C_VEL
LIN {X 0,Y 734.603,Z 1008.259,A -85,B 0,C 180,E1 1679.327,E2 1679.327} C_VEL
LIN {X 0,Y 732.912,Z 1073.474,A -85,B 0,C 180,E1 1683.911,E2 1683.911} C_VEL
LIN {X 0,Y 731.667,Z 1126.044,A -85,B 0,C 180,E1 1689.079,E2 1689.079} C_VEL
LIN {X 0,Y 731.172,Z 1162.482,A -85,B 0,C 180,E1 1694.048,E2 1694.048} C_VEL
LIN {X 0,Y 731.033,Z 1188.72,A -85,B 0,C 180,E1 1699.238,E2 1699.238} C_VEL
LIN {X 0,Y 731.12,Z 1204.76,A -85,B 0,C 180,E1 1704.643,E2 1704.643} C_VEL
LIN {X 0,Y 730.991,Z 1209.838,A -85,B 0,C 180,E1 1710.593,E2 1710.593} C_VEL
LIN {X 0,Y 731.124,Z 1203.526,A -85,B 0,C 180,E1 1715.952,E2 1715.952} C_VEL
LIN {X 0,Y 731.285,Z 1184.861,A -85,B 0,C 180,E1 1721.664,E2 1721.664} C_VEL
LIN {X 0,Y 731.524,Z 1152.422,A -85,B 0,C 180,E1 1727.492,E2 1727.492} C_VEL
LIN {X 0,Y 732.467,Z 1106.374,A -85,B 0,C 180,E1 1733.053,E2 1733.053} C_VEL
LIN {X 0,Y 733.722,Z 1047.809,A -85,B 0,C 180,E1 1738.077,E2 1738.077} C_VEL
LIN {X 0,Y 735.274,Z 978.852,A -85,B 0,C 180,E1 1742.264,E2 1742.264} C_VEL
LIN {X 0,Y 736.743,Z 906.556,A -85,B 0,C 180,E1 1745.196,E2 1745.196} C_VEL
LIN {X 0,Y 737.576,Z 832.685,A -85,B 0,C 180,E1 1746.935,E2 1746.935} C_VEL
LIN {X 0,Y 735.749,Z 772.126,A -85,B 0,C 180,E1 1747.806,E2 1747.806} C_VEL
LIN {X 0,Y 731.077,Z 762.06,A -85,B 0,C 180,E1 1748.41,E2 1748.41} C_VEL
LIN {X 0,Y 730.511,Z 762.06,A -85,B 0,C 180,E1 1754.19,E2 1754.19} C_VEL
LIN {X 0,Y 730.787,Z 762.06,A -85,B 0,C 180,E1 1762.2,E2 1762.2} C_VEL
LIN {X 0,Y 730.893,Z 762.06,A -85,B 0,C 180,E1 1768.011,E2 1768.011} C_VEL
LIN {X 0,Y 730.876,Z 762.06,A -85,B 0,C 180,E1 1774.79,E2 1774.79} C_VEL
LIN {X 0,Y 731.205,Z 762.06,A -85,B 0,C 180,E1 1782.47,E2 1782.47} C_VEL
LIN {X 0,Y 730.845,Z 762.06,A -85,B 0,C 180,E1 1791.027,E2 1791.027} C_VEL
LIN {X 0,Y 731.079,Z 762.06,A -85,B 0,C 180,E1 1798.203,E2 1798.203} C_VEL
LIN {X 0,Y 731.318,Z 762.06,A -85,B 0,C 180,E1 1805.347,E2 1805.347} C_VEL
LIN {X 0,Y 730.721,Z 762.06,A -85,B 0,C 180,E1 1813.807,E2 1813.807} C_VEL
LIN {X 0,Y 730.834,Z 762.06,A -85,B 0,C 180,E1 1821.299,E2 1821.299} C_VEL
LIN {X 0,Y 731.146,Z 762.06,A -85,B 0,C 180,E1 1829.185,E2 1829.185} C_VEL
LIN {X 0,Y 730.592,Z 762.06,A -85,B 0,C 180,E1 1836.952,E2 1836.952} C_VEL
LIN {X 0,Y 730.492,Z 762.06,A -85,B 0,C 180,E1 1844.258,E2 1844.258} C_VEL
LIN {X 0,Y 730.853,Z 762.06,A -85,B 0,C 180,E1 1852.258,E2 1852.258} C_VEL
LIN {X 0,Y 731.294,Z 763.832,A -85,B 0,C 180,E1 1855.406,E2 1855.406} C_VEL
LIN {X 0,Y 736.018,Z 778.771,A -85,B 0,C 180,E1 1855.832,E2 1855.832} C_VEL
LIN {X 0,Y 736.367,Z 869.244,A -85,B 0,C 180,E1 1857.191,E2 1857.191} C_VEL
LIN {X 0,Y 735.281,Z 938.962,A -85,B 0,C 180,E1 1859.37,E2 1859.37} C_VEL
LIN {X 0,Y 733.858,Z 1007.206,A -85,B 0,C 180,E1 1862.804,E2 1862.804} C_VEL
LIN {X 0,Y 732.465,Z 1066.74,A -85,B 0,C 180,E1 1867.207,E2 1867.207} C_VEL
LIN {X 0,Y 731.528,Z 1114.055,A -85,B 0,C 180,E1 1872.196,E2 1872.196} C_VEL
LIN {X 0,Y 730.902,Z 1146.777,A -85,B 0,C 180,E1 1877.168,E2 1877.168} C_VEL
LIN {X 0,Y 731.11,Z 1166.127,A -85,B 0,C 180,E1 1881.652,E2 1881.652} C_VEL
LIN {X 0,Y 731.062,Z 1178.298,A -85,B 0,C 180,E1 1887.029,E2 1887.029} C_VEL
LIN {X 0,Y 731.275,Z 1179.262,A -85,B 0,C 180,E1 1891.784,E2 1891.784} C_VEL
LIN {X 0,Y 731.329,Z 1167.764,A -85,B 0,C 180,E1 1897.747,E2 1897.747} C_VEL
LIN {X 0,Y 731.38,Z 1141.799,A -85,B 0,C 180,E1 1903.622,E2 1903.622} C_VEL
LIN {X 0,Y 731.986,Z 1102.849,A -85,B 0,C 180,E1 1909.06,E2 1909.06} C_VEL
LIN {X 0,Y 733.019,Z 1050.317,A -85,B 0,C 180,E1 1914.081,E2 1914.081} C_VEL
LIN {X 0,Y 734.339,Z 986.804,A -85,B 0,C 180,E1 1918.281,E2 1918.281} C_VEL
LIN {X 0,Y 735.737,Z 917.071,A -85,B 0,C 180,E1 1921.353,E2 1921.353} C_VEL
LIN {X 0,Y 736.645,Z 846.634,A -85,B 0,C 180,E1 1923.168,E2 1923.168} C_VEL
LIN {X 0,Y 733.792,Z 767.705,A -85,B 0,C 180,E1 1924.324,E2 1924.324} C_VEL
LIN {X 0,Y 731.513,Z 762.06,A -85,B 0,C 180,E1 1924.591,E2 1924.591} C_VEL
LIN {X 0,Y 730.98,Z 762.06,A -85,B 0,C 180,E1 1934.263,E2 1934.263} C_VEL
LIN {X 0,Y 730.821,Z 762.06,A -85,B 0,C 180,E1 1943.723,E2 1943.723} C_VEL
LIN {X 0,Y 730.731,Z 762.06,A -85,B 0,C 180,E1 1951.889,E2 1951.889} C_VEL
LIN {X 0,Y 731.026,Z 762.06,A -85,B 0,C 180,E1 1958.707,E2 1958.707} C_VEL
LIN {X 0,Y 731.381,Z 762.06,A -85,B 0,C 180,E1 1967.427,E2 1967.427} C_VEL
LIN {X 0,Y 731.739,Z 762.06,A -85,B 0,C 180,E1 1977.04,E2 1977.04} C_VEL
LIN {X 0,Y 731.288,Z 762.06,A -85,B 0,C 180,E1 1985.371,E2 1985.371} C_VEL
LIN {X 0,Y 730.335,Z 762.06,A -85,B 0,C 180,E1 1987.348,E2 1987.348} C_VEL
LIN {X 0,Y 722.488,Z 762.06,A -85,B 0,C 180,E1 1990.081,E2 1990.081} C_VEL
LIN {X 0,Y 722.226,Z 762.06,A -85,B 0,C 180,E1 1995.243,E2 1995.243} C_VEL
LIN {X 0,Y 722.695,Z 762.06,A -85,B 0,C 180,E1 2001.577,E2 2001.577} C_VEL
LIN {X 0,Y 722.846,Z 762.06,A -85,B 0,C 180,E1 2009.581,E2 2009.581} C_VEL
LIN {X 0,Y 722.395,Z 762.06,A -85,B 0,C 180,E1 2018.318,E2 2018.318} C_VEL
LIN {X 0,Y 722.639,Z 762.06,A -85,B 0,C 180,E1 2026.456,E2 2026.456} C_VEL
LIN {X 0,Y 722.449,Z 763.572,A -85,B 0,C 180,E1 2031.264,E2 2031.264} C_VEL
LIN {X 0,Y 731.122,Z 782.32,A -85,B 0,C 180,E1 2032.037,E2 2032.037} C_VEL
LIN {X 0,Y 730.842,Z 869.043,A -85,B 0,C 180,E1 2033.396,E2 2033.396} C_VEL
LIN {X 0,Y 729.343,Z 939.538,A -85,B 0,C 180,E1 2035.615,E2 2035.615} C_VEL
LIN {X 0,Y 727.369,Z 1009.817,A -85,B 0,C 180,E1 2039.086,E2 2039.086} C_VEL
LIN {X 0,Y 725.372,Z 1073.963,A -85,B 0,C 180,E1 2043.661,E2 2043.661} C_VEL
LIN {X 0,Y 723.941,Z 1125.478,A -85,B 0,C 180,E1 2048.777,E2 2048.777} C_VEL
LIN {X 0,Y 723.292,Z 1162.479,A -85,B 0,C 180,E1 2053.869,E2 2053.869} C_VEL
LIN {X 0,Y 722.968,Z 1189.929,A -85,B 0,C 180,E1 2059.423,E2 2059.423} C_VEL
LIN {X 0,Y 723.151,Z 1204.76,A -85,B 0,C 180,E1 2064.584,E2 2064.584} C_VEL
LIN {X 0,Y 722.985,Z 1209.838,A -85,B 0,C 180,E1 2070.6,E2 2070.6} C_VEL
LIN {X 0,Y 723.113,Z 1203.526,A -85,B 0,C 180,E1 2076.018,E2 2076.018} C_VEL
LIN {X 0,Y 723.162,Z 1184.043,A -85,B 0,C 180,E1 2081.982,E2 2081.982} C_VEL
LIN {X 0,Y 723.579,Z 1152.423,A -85,B 0,C 180,E1 2087.691,E2 2087.691} C_VEL
LIN {X 0,Y 724.704,Z 1105.269,A -85,B 0,C 180,E1 2093.426,E2 2093.426} C_VEL
LIN {X 0,Y 726.299,Z 1046.866,A -85,B 0,C 180,E1 2098.46,E2 2098.46} C_VEL
LIN {X 0,Y 728.332,Z 978.033,A -85,B 0,C 180,E1 2102.652,E2 2102.652} C_VEL
LIN {X 0,Y 730.094,Z 906.414,A -85,B 0,C 180,E1 2105.57,E2 2105.57} C_VEL
LIN {X 0,Y 731.199,Z 832.196,A -85,B 0,C 180,E1 2107.319,E2 2107.319} C_VEL
LIN {X 0,Y 729.757,Z 775.997,A -85,B 0,C 180,E1 2108.124,E2 2108.124} C_VEL
LIN {X 0,Y 723.022,Z 762.06,A -85,B 0,C 180,E1 2108.813,E2 2108.813} C_VEL
LIN {X 0,Y 722.158,Z 762.06,A -85,B 0,C 180,E1 2115.227,E2 2115.227} C_VEL
LIN {X 0,Y 722.879,Z 762.06,A -85,B 0,C 180,E1 2121.877,E2 2121.877} C_VEL
LIN {X 0,Y 722.585,Z 762.06,A -85,B 0,C 180,E1 2129.013,E2 2129.013} C_VEL
LIN {X 0,Y 722.402,Z 762.06,A -85,B 0,C 180,E1 2135.945,E2 2135.945} C_VEL
LIN {X 0,Y 722.664,Z 762.06,A -85,B 0,C 180,E1 2143.516,E2 2143.516} C_VEL
LIN {X 0,Y 722.9,Z 762.06,A -85,B 0,C 180,E1 2150.927,E2 2150.927} C_VEL
LIN {X 0,Y 723.083,Z 762.06,A -85,B 0,C 180,E1 2158.183,E2 2158.183} C_VEL
LIN {X 0,Y 723.277,Z 762.06,A -85,B 0,C 180,E1 2165.406,E2 2165.406} C_VEL
LIN {X 0,Y 722.638,Z 762.06,A -85,B 0,C 180,E1 2173.965,E2 2173.965} C_VEL
LIN {X 0,Y 722.676,Z 762.06,A -85,B 0,C 180,E1 2181.551,E2 2181.551} C_VEL
LIN {X 0,Y 722.983,Z 762.06,A -85,B 0,C 180,E1 2189.547,E2 2189.547} C_VEL
LIN {X 0,Y 722.662,Z 762.06,A -85,B 0,C 180,E1 2196.753,E2 2196.753} C_VEL
LIN {X 0,Y 722.713,Z 762.06,A -85,B 0,C 180,E1 2203.622,E2 2203.622} C_VEL
LIN {X 0,Y 722.922,Z 762.06,A -85,B 0,C 180,E1 2211.916,E2 2211.916} C_VEL
LIN {X 0,Y 723.178,Z 764.071,A -85,B 0,C 180,E1 2214.965,E2 2214.965} C_VEL
LIN {X 0,Y 729.39,Z 778.972,A -85,B 0,C 180,E1 2215.481,E2 2215.481} C_VEL
LIN {X 0,Y 729.577,Z 871.182,A -85,B 0,C 180,E1 2216.891,E2 2216.891} C_VEL
LIN {X 0,Y 728.221,Z 940.68,A -85,B 0,C 180,E1 2219.112,E2 2219.112} C_VEL
LIN {X 0,Y 726.472,Z 1008.591,A -85,B 0,C 180,E1 2222.589,E2 2222.589} C_VEL
LIN {X 0,Y 724.779,Z 1068.233,A -85,B 0,C 180,E1 2227.09,E2 2227.09} C_VEL
LIN {X 0,Y 723.638,Z 1115.272,A -85,B 0,C 180,E1 2232.153,E2 2232.153} C_VEL
LIN {X 0,Y 722.972,Z 1146.498,A -85,B 0,C 180,E1 2236.969,E2 2236.969} C_VEL
LIN {X 0,Y 722.928,Z 1168.061,A -85,B 0,C 180,E1 2242.164,E2 2242.164} C_VEL
LIN {X 0,Y 723.071,Z 1178.297,A -85,B 0,C 180,E1 2246.996,E2 2246.996} C_VEL
LIN {X 0,Y 723.266,Z 1179.262,A -85,B 0,C 180,E1 2251.804,E2 2251.804} C_VEL
LIN {X 0,Y 723.286,Z 1167.766,A -85,B 0,C 180,E1 2257.834,E2 2257.834} C_VEL
LIN {X 0,Y 723.438,Z 1142.496,A -85,B 0,C 180,E1 2263.653,E2 2263.653} C_VEL
LIN {X 0,Y 724.134,Z 1102.855,A -85,B 0,C 180,E1 2269.275,E2 2269.275} C_VEL
LIN {X 0,Y 725.388,Z 1050.348,A -85,B 0,C 180,E1 2274.348,E2 2274.348} C_VEL
LIN {X 0,Y 727.051,Z 987.584,A -85,B 0,C 180,E1 2278.548,E2 2278.548} C_VEL
LIN {X 0,Y 728.76,Z 918.588,A -85,B 0,C 180,E1 2281.634,E2 2281.634} C_VEL
LIN {X 0,Y 729.884,Z 848.613,A -85,B 0,C 180,E1 2283.48,E2 2283.48} C_VEL
LIN {X 0,Y 727.605,Z 771.706,A -85,B 0,C 180,E1 2284.611,E2 2284.611} C_VEL
LIN {X 0,Y 723.46,Z 762.06,A -85,B 0,C 180,E1 2284.962,E2 2284.962} C_VEL
LIN {X 0,Y 722.938,Z 762.06,A -85,B 0,C 180,E1 2295.323,E2 2295.323} C_VEL
LIN {X 0,Y 722.744,Z 762.06,A -85,B 0,C 180,E1 2303.887,E2 2303.887} C_VEL
LIN {X 0,Y 722.775,Z 762.06,A -85,B 0,C 180,E1 2311.818,E2 2311.818} C_VEL
LIN {X 0,Y 722.594,Z 762.06,A -85,B 0,C 180,E1 2319.735,E2 2319.735} C_VEL
LIN {X 0,Y 723.371,Z 762.06,A -85,B 0,C 180,E1 2327.285,E2 2327.285} C_VEL
LIN {X 0,Y 723.699,Z 762.06,A -85,B 0,C 180,E1 2337.007,E2 2337.007} C_VEL
LIN {X 0,Y 723.249,Z 762.06,A -85,B 0,C 180,E1 2345.431,E2 2345.431} C_VEL
LIN {X 0,Y 722.488,Z 762.06,A -85,B 0,C 180,E1 2350.081,E2 2350.081} C_VEL
LIN {X 0,Y 715.243,Z 762.06,A -85,B 0,C 180,E1 2352.86,E2 2352.86} C_VEL
LIN {X 0,Y 714.544,Z 762.06,A -85,B 0,C 180,E1 2361.836,E2 2361.836} C_VEL
LIN {X 0,Y 714.638,Z 762.06,A -85,B 0,C 180,E1 2369.956,E2 2369.956} C_VEL
LIN {X 0,Y 714.719,Z 762.06,A -85,B 0,C 180,E1 2377.278,E2 2377.278} C_VEL
LIN {X 0,Y 714.667,Z 762.06,A -85,B 0,C 180,E1 2386.396,E2 2386.396} C_VEL
LIN {X 0,Y 714.349,Z 763.836,A -85,B 0,C 180,E1 2390.745,E2 2390.745} C_VEL
LIN {X 0,Y 724.818,Z 785.527,A -85,B 0,C 180,E1 2391.687,E2 2391.687} C_VEL
LIN {X 0,Y 724.34,Z 869.985,A -85,B 0,C 180,E1 2393.037,E2 2393.037} C_VEL
LIN {X 0,Y 722.56,Z 940.253,A -85,B 0,C 180,E1 2395.277,E2 2395.277} C_VEL
LIN {X 0,Y 720.159,Z 1011.754,A -85,B 0,C 180,E1 2398.865,E2 2398.865} C_VEL
LIN {X 0,Y 717.776,Z 1076.521,A -85,B 0,C 180,E1 2403.585,E2 2403.585} C_VEL
LIN {X 0,Y 716.098,Z 1127.85,A -85,B 0,C 180,E1 2408.82,E2 2408.82} C_VEL
LIN {X 0,Y 715.29,Z 1164.372,A -85,B 0,C 180,E1 2414,E2 2414} C_VEL
LIN {X 0,Y 715.031,Z 1189.927,A -85,B 0,C 180,E1 2419.304,E2 2419.304} C_VEL
LIN {X 0,Y 714.916,Z 1205.881,A -85,B 0,C 180,E1 2425.131,E2 2425.131} C_VEL
LIN {X 0,Y 714.987,Z 1209.838,A -85,B 0,C 180,E1 2430.606,E2 2430.606} C_VEL
LIN {X 0,Y 715.109,Z 1203.526,A -85,B 0,C 180,E1 2436.085,E2 2436.085} C_VEL
LIN {X 0,Y 715.365,Z 1186.216,A -85,B 0,C 180,E1 2441.617,E2 2441.617} C_VEL
LIN {X 0,Y 715.687,Z 1153.899,A -85,B 0,C 180,E1 2447.676,E2 2447.676} C_VEL
LIN {X 0,Y 717.004,Z 1106.88,A -85,B 0,C 180,E1 2453.528,E2 2453.528} C_VEL
LIN {X 0,Y 718.898,Z 1047.69,A -85,B 0,C 180,E1 2458.718,E2 2458.718} C_VEL
LIN {X 0,Y 721.309,Z 979.503,A -85,B 0,C 180,E1 2462.932,E2 2462.932} C_VEL
LIN {X 0,Y 723.428,Z 908.13,A -85,B 0,C 180,E1 2465.891,E2 2465.891} C_VEL
LIN {X 0,Y 724.767,Z 834.672,A -85,B 0,C 180,E1 2467.669,E2 2467.669} C_VEL
LIN {X 0,Y 723.35,Z 778.737,A -85,B 0,C 180,E1 2468.49,E2 2468.49} C_VEL
LIN {X 0,Y 715.007,Z 762.06,A -85,B 0,C 180,E1 2469.292,E2 2469.292} C_VEL
LIN {X 0,Y 714.046,Z 762.06,A -85,B 0,C 180,E1 2476.287,E2 2476.287} C_VEL
LIN {X 0,Y 714.669,Z 762.06,A -85,B 0,C 180,E1 2482.735,E2 2482.735} C_VEL
LIN {X 0,Y 714.459,Z 762.06,A -85,B 0,C 180,E1 2490.036,E2 2490.036} C_VEL
LIN {X 0,Y 714.113,Z 762.06,A -85,B 0,C 180,E1 2496.832,E2 2496.832} C_VEL
LIN {X 0,Y 714.755,Z 762.06,A -85,B 0,C 180,E1 2503.328,E2 2503.328} C_VEL
LIN {X 0,Y 714.923,Z 762.06,A -85,B 0,C 180,E1 2510.825,E2 2510.825} C_VEL
LIN {X 0,Y 715.086,Z 762.06,A -85,B 0,C 180,E1 2518.163,E2 2518.163} C_VEL
LIN {X 0,Y 715.225,Z 762.06,A -85,B 0,C 180,E1 2525.467,E2 2525.467} C_VEL
LIN {X 0,Y 715.226,Z 762.06,A -85,B 0,C 180,E1 2532.862,E2 2532.862} C_VEL
LIN {X 0,Y 714.53,Z 762.06,A -85,B 0,C 180,E1 2541.809,E2 2541.809} C_VEL
LIN {X 0,Y 714.84,Z 762.06,A -85,B 0,C 180,E1 2549.917,E2 2549.917} C_VEL
LIN {X 0,Y 714.507,Z 762.06,A -85,B 0,C 180,E1 2557.26,E2 2557.26} C_VEL
LIN {X 0,Y 714.705,Z 762.06,A -85,B 0,C 180,E1 2563.628,E2 2563.628} C_VEL
LIN {X 0,Y 714.967,Z 762.06,A -85,B 0,C 180,E1 2571.266,E2 2571.266} C_VEL
LIN {X 0,Y 715.043,Z 764.04,A -85,B 0,C 180,E1 2574.507,E2 2574.507} C_VEL
LIN {X 0,Y 722.853,Z 782.736,A -85,B 0,C 180,E1 2575.169,E2 2575.169} C_VEL
LIN {X 0,Y 722.813,Z 871.789,A -85,B 0,C 180,E1 2576.555,E2 2576.555} C_VEL
LIN {X 0,Y 721.192,Z 941.215,A -85,B 0,C 180,E1 2578.8,E2 2578.8} C_VEL
LIN {X 0,Y 719.065,Z 1008.584,A -85,B 0,C 180,E1 2582.283,E2 2582.283} C_VEL
LIN {X 0,Y 717.132,Z 1067.962,A -85,B 0,C 180,E1 2586.806,E2 2586.806} C_VEL
LIN {X 0,Y 715.814,Z 1115.27,A -85,B 0,C 180,E1 2591.952,E2 2591.952} C_VEL
LIN {X 0,Y 715.04,Z 1146.496,A -85,B 0,C 180,E1 2596.822,E2 2596.822} C_VEL
LIN {X 0,Y 714.96,Z 1168.06,A -85,B 0,C 180,E1 2602.076,E2 2602.076} C_VEL
LIN {X 0,Y 715.11,Z 1178.297,A -85,B 0,C 180,E1 2606.962,E2 2606.962} C_VEL
LIN {X 0,Y 715.257,Z 1179.263,A -85,B 0,C 180,E1 2611.824,E2 2611.824} C_VEL
LIN {X 0,Y 715.249,Z 1167.768,A -85,B 0,C 180,E1 2617.923,E2 2617.923} C_VEL
LIN {X 0,Y 715.441,Z 1142.563,A -85,B 0,C 180,E1 2623.797,E2 2623.797} C_VEL
LIN {X 0,Y 716.281,Z 1103.824,A -85,B 0,C 180,E1 2629.379,E2 2629.379} C_VEL
LIN {X 0,Y 717.758,Z 1052.11,A -85,B 0,C 180,E1 2634.478,E2 2634.478} C_VEL
LIN {X 0,Y 719.768,Z 989.68,A -85,B 0,C 180,E1 2638.746,E2 2638.746} C_VEL
LIN {X 0,Y 721.761,Z 921.097,A -85,B 0,C 180,E1 2641.885,E2 2641.885} C_VEL
LIN {X 0,Y 723.166,Z 850.518,A -85,B 0,C 180,E1 2643.799,E2 2643.799} C_VEL
LIN {X 0,Y 721.034,Z 774.792,A -85,B 0,C 180,E1 2644.936,E2 2644.936} C_VEL
LIN {X 0,Y 715.344,Z 762.06,A -85,B 0,C 180,E1 2645.481,E2 2645.481} C_VEL
LIN {X 0,Y 714.937,Z 762.06,A -85,B 0,C 180,E1 2655.285,E2 2655.285} C_VEL
LIN {X 0,Y 714.617,Z 762.06,A -85,B 0,C 180,E1 2664.277,E2 2664.277} C_VEL
LIN {X 0,Y 714.816,Z 762.06,A -85,B 0,C 180,E1 2671.698,E2 2671.698} C_VEL
LIN {X 0,Y 714.686,Z 762.06,A -85,B 0,C 180,E1 2679.501,E2 2679.501} C_VEL
LIN {X 0,Y 715.404,Z 762.06,A -85,B 0,C 180,E1 2687.141,E2 2687.141} C_VEL
LIN {X 0,Y 715.658,Z 762.06,A -85,B 0,C 180,E1 2696.973,E2 2696.973} C_VEL
LIN {X 0,Y 715.198,Z 762.06,A -85,B 0,C 180,E1 2705.493,E2 2705.493} C_VEL
LIN {X 0,Y 715.243,Z 762.06,A -85,B 0,C 180,E1 2712.86,E2 2712.86} C_VEL
LIN {X 0,Y 706.165,Z 762.06,A -85,B 0,C 180,E1 2715.624,E2 2715.624} C_VEL
LIN {X 0,Y 706.438,Z 762.06,A -85,B 0,C 180,E1 2722.099,E2 2722.099} C_VEL
LIN {X 0,Y 706.692,Z 762.06,A -85,B 0,C 180,E1 2729.643,E2 2729.643} C_VEL
LIN {X 0,Y 706.505,Z 762.06,A -85,B 0,C 180,E1 2737.77,E2 2737.77} C_VEL
LIN {X 0,Y 706.741,Z 762.06,A -85,B 0,C 180,E1 2746.027,E2 2746.027} C_VEL
LIN {X 0,Y 706.198,Z 763.936,A -85,B 0,C 180,E1 2750.203,E2 2750.203} C_VEL
LIN {X 0,Y 718.506,Z 787.988,A -85,B 0,C 180,E1 2751.319,E2 2751.319} C_VEL
LIN {X 0,Y 717.856,Z 871.696,A -85,B 0,C 180,E1 2752.69,E2 2752.69} C_VEL
LIN {X 0,Y 715.697,Z 943.213,A -85,B 0,C 180,E1 2755.024,E2 2755.024} C_VEL
LIN {X 0,Y 712.905,Z 1014.163,A -85,B 0,C 180,E1 2758.668,E2 2758.668} C_VEL
LIN {X 0,Y 710.211,Z 1078.489,A -85,B 0,C 180,E1 2763.457,E2 2763.457} C_VEL
LIN {X 0,Y 708.244,Z 1129.864,A -85,B 0,C 180,E1 2768.819,E2 2768.819} C_VEL
LIN {X 0,Y 707.433,Z 1164.374,A -85,B 0,C 180,E1 2773.817,E2 2773.817} C_VEL
LIN {X 0,Y 706.975,Z 1191.07,A -85,B 0,C 180,E1 2779.493,E2 2779.493} C_VEL
LIN {X 0,Y 706.964,Z 1205.88,A -85,B 0,C 180,E1 2785.076,E2 2785.076} C_VEL
LIN {X 0,Y 706.981,Z 1209.838,A -85,B 0,C 180,E1 2790.613,E2 2790.613} C_VEL
LIN {X 0,Y 707.103,Z 1203.526,A -85,B 0,C 180,E1 2796.155,E2 2796.155} C_VEL
LIN {X 0,Y 707.187,Z 1184.933,A -85,B 0,C 180,E1 2802.051,E2 2802.051} C_VEL
LIN {X 0,Y 707.782,Z 1153.918,A -85,B 0,C 180,E1 2807.876,E2 2807.876} C_VEL
LIN {X 0,Y 709.277,Z 1108.658,A -85,B 0,C 180,E1 2813.614,E2 2813.614} C_VEL
LIN {X 0,Y 711.468,Z 1049.734,A -85,B 0,C 180,E1 2818.891,E2 2818.891} C_VEL
LIN {X 0,Y 714.295,Z 981.337,A -85,B 0,C 180,E1 2823.199,E2 2823.199} C_VEL
LIN {X 0,Y 716.811,Z 909.431,A -85,B 0,C 180,E1 2826.231,E2 2826.231} C_VEL
LIN {X 0,Y 718.428,Z 835.204,A -85,B 0,C 180,E1 2828.052,E2 2828.052} C_VEL
LIN {X 0,Y 717.065,Z 782.034,A -85,B 0,C 180,E1 2828.849,E2 2828.849} C_VEL
LIN {X 0,Y 707.015,Z 762.06,A -85,B 0,C 180,E1 2829.816,E2 2829.816} C_VEL
LIN {X 0,Y 706.261,Z 762.06,A -85,B 0,C 180,E1 2837.798,E2 2837.798} C_VEL
LIN {X 0,Y 706.986,Z 762.06,A -85,B 0,C 180,E1 2845.671,E2 2845.671} C_VEL
LIN {X 0,Y 706.973,Z 762.06,A -85,B 0,C 180,E1 2853.875,E2 2853.875} C_VEL
LIN {X 0,Y 706.792,Z 762.06,A -85,B 0,C 180,E1 2863.134,E2 2863.134} C_VEL
LIN {X 0,Y 706.96,Z 762.06,A -85,B 0,C 180,E1 2870.721,E2 2870.721} C_VEL
LIN {X 0,Y 707.09,Z 762.06,A -85,B 0,C 180,E1 2878.142,E2 2878.142} C_VEL
LIN {X 0,Y 707.195,Z 762.06,A -85,B 0,C 180,E1 2885.53,E2 2885.53} C_VEL
LIN {X 0,Y 707.143,Z 762.06,A -85,B 0,C 180,E1 2893.012,E2 2893.012} C_VEL
LIN {X 0,Y 706.785,Z 762.06,A -85,B 0,C 180,E1 2901.039,E2 2901.039} C_VEL
LIN {X 0,Y 706.753,Z 762.06,A -85,B 0,C 180,E1 2910.295,E2 2910.295} C_VEL
LIN {X 0,Y 706.742,Z 762.06,A -85,B 0,C 180,E1 2916.424,E2 2916.424} C_VEL
LIN {X 0,Y 706.464,Z 762.06,A -85,B 0,C 180,E1 2924.269,E2 2924.269} C_VEL
LIN {X 0,Y 706.787,Z 762.06,A -85,B 0,C 180,E1 2932.303,E2 2932.303} C_VEL
LIN {X 0,Y 706.917,Z 763.708,A -85,B 0,C 180,E1 2934.033,E2 2934.033} C_VEL
LIN {X 0,Y 716.268,Z 783.072,A -85,B 0,C 180,E1 2934.806,E2 2934.806} C_VEL
LIN {X 0,Y 716.093,Z 872.202,A -85,B 0,C 180,E1 2936.209,E2 2936.209} C_VEL
LIN {X 0,Y 714.164,Z 942.364,A -85,B 0,C 180,E1 2938.506,E2 2938.506} C_VEL
LIN {X 0,Y 711.72,Z 1009.216,A -85,B 0,C 180,E1 2942.014,E2 2942.014} C_VEL
LIN {X 0,Y 709.494,Z 1067.956,A -85,B 0,C 180,E1 2946.542,E2 2946.542} C_VEL
LIN {X 0,Y 707.964,Z 1115.267,A -85,B 0,C 180,E1 2951.744,E2 2951.744} C_VEL
LIN {X 0,Y 707.057,Z 1148.046,A -85,B 0,C 180,E1 2956.986,E2 2956.986} C_VEL
LIN {X 0,Y 707.025,Z 1168.058,A -85,B 0,C 180,E1 2961.987,E2 2961.987} C_VEL
LIN {X 0,Y 707.118,Z 1178.296,A -85,B 0,C 180,E1 2966.928,E2 2966.928} C_VEL
LIN {X 0,Y 707.248,Z 1179.263,A -85,B 0,C 180,E1 2971.844,E2 2971.844} C_VEL
LIN {X 0,Y 707.228,Z 1167.77,A -85,B 0,C 180,E1 2978.013,E2 2978.013} C_VEL
LIN {X 0,Y 707.551,Z 1144.32,A -85,B 0,C 180,E1 2983.638,E2 2983.638} C_VEL
LIN {X 0,Y 708.441,Z 1105.675,A -85,B 0,C 180,E1 2989.379,E2 2989.379} C_VEL
LIN {X 0,Y 710.138,Z 1053.804,A -85,B 0,C 180,E1 2994.61,E2 2994.61} C_VEL
LIN {X 0,Y 712.476,Z 991.952,A -85,B 0,C 180,E1 2998.939,E2 2998.939} C_VEL
LIN {X 0,Y 714.79,Z 923.755,A -85,B 0,C 180,E1 3002.135,E2 3002.135} C_VEL
LIN {X 0,Y 716.492,Z 852.571,A -85,B 0,C 180,E1 3004.119,E2 3004.119} C_VEL
LIN {X 0,Y 714.572,Z 777.616,A -85,B 0,C 180,E1 3005.266,E2 3005.266} C_VEL
LIN {X 0,Y 707.185,Z 762.06,A -85,B 0,C 180,E1 3005.97,E2 3005.97} C_VEL
LIN {X 0,Y 706.762,Z 762.06,A -85,B 0,C 180,E1 3015.959,E2 3015.959} C_VEL
LIN {X 0,Y 706.646,Z 762.06,A -85,B 0,C 180,E1 3023.811,E2 3023.811} C_VEL
LIN {X 0,Y 706.813,Z 762.06,A -85,B 0,C 180,E1 3031.122,E2 3031.122} C_VEL
LIN {X 0,Y 706.72,Z 762.06,A -85,B 0,C 180,E1 3039.259,E2 3039.259} C_VEL
LIN {X 0,Y 707.396,Z 762.06,A -85,B 0,C 180,E1 3047.277,E2 3047.277} C_VEL
LIN {X 0,Y 707.615,Z 762.06,A -85,B 0,C 180,E1 3056.945,E2 3056.945} C_VEL
LIN {X 0,Y 707.16,Z 762.06,A -85,B 0,C 180,E1 3065.555,E2 3065.555} C_VEL
LIN {X 0,Y 707.139,Z 762.06,A -85,B 0,C 180,E1 3073.038,E2 3073.038} C_VEL
LIN {X 0,Y 706.165,Z 762.06,A -85,B 0,C 180,E1 3075.624,E2 3075.624} C_VEL
LIN {X 0,Y 698.58,Z 762.06,A -85,B 0,C 180,E1 3078.448,E2 3078.448} C_VEL
LIN {X 0,Y 698.408,Z 762.06,A -85,B 0,C 180,E1 3086.47,E2 3086.47} C_VEL
LIN {X 0,Y 698.159,Z 762.06,A -85,B 0,C 180,E1 3093.683,E2 3093.683} C_VEL
LIN {X 0,Y 697.866,Z 762.06,A -85,B 0,C 180,E1 3099.928,E2 3099.928} C_VEL
LIN {X 0,Y 698.38,Z 762.06,A -85,B 0,C 180,E1 3106.84,E2 3106.84} C_VEL
LIN {X 0,Y 698.031,Z 763.385,A -85,B 0,C 180,E1 3109.635,E2 3109.635} C_VEL
LIN {X 0,Y 712.23,Z 790.535,A -85,B 0,C 180,E1 3110.946,E2 3110.946} C_VEL
LIN {X 0,Y 711.409,Z 873.258,A -85,B 0,C 180,E1 3112.333,E2 3112.333} C_VEL
LIN {X 0,Y 708.938,Z 943.886,A -85,B 0,C 180,E1 3114.671,E2 3114.671} C_VEL
LIN {X 0,Y 705.801,Z 1014.553,A -85,B 0,C 180,E1 3118.342,E2 3118.342} C_VEL
LIN {X 0,Y 702.672,Z 1079.289,A -85,B 0,C 180,E1 3123.221,E2 3123.221} C_VEL
LIN {X 0,Y 700.522,Z 1129.866,A -85,B 0,C 180,E1 3128.574,E2 3128.574} C_VEL
LIN {X 0,Y 699.411,Z 1166.14,A -85,B 0,C 180,E1 3133.95,E2 3133.95} C_VEL
LIN {X 0,Y 699.03,Z 1191.069,A -85,B 0,C 180,E1 3139.372,E2 3139.372} C_VEL
LIN {X 0,Y 699.003,Z 1205.88,A -85,B 0,C 180,E1 3145.02,E2 3145.02} C_VEL
LIN {X 0,Y 698.992,Z 1209.838,A -85,B 0,C 180,E1 3150.62,E2 3150.62} C_VEL
LIN {X 0,Y 699.087,Z 1203.526,A -85,B 0,C 180,E1 3156.226,E2 3156.226} C_VEL
LIN {X 0,Y 699.201,Z 1184.935,A -85,B 0,C 180,E1 3162.191,E2 3162.191} C_VEL
LIN {X 0,Y 699.834,Z 1153.628,A -85,B 0,C 180,E1 3168.13,E2 3168.13} C_VEL
LIN {X 0,Y 701.572,Z 1107.565,A -85,B 0,C 180,E1 3174.005,E2 3174.005} C_VEL
LIN {X 0,Y 704.187,Z 1048.47,A -85,B 0,C 180,E1 3179.316,E2 3179.316} C_VEL
LIN {X 0,Y 707.374,Z 980.686,A -85,B 0,C 180,E1 3183.602,E2 3183.602} C_VEL
LIN {X 0,Y 710.264,Z 909.593,A -85,B 0,C 180,E1 3186.614,E2 3186.614} C_VEL
LIN {X 0,Y 712.16,Z 834.887,A -85,B 0,C 180,E1 3188.453,E2 3188.453} C_VEL
LIN {X 0,Y 710.771,Z 785.058,A -85,B 0,C 180,E1 3189.22,E2 3189.22} C_VEL
LIN {X 0,Y 699.049,Z 762.06,A -85,B 0,C 180,E1 3190.434,E2 3190.434} C_VEL
LIN {X 0,Y 698.891,Z 762.06,A -85,B 0,C 180,E1 3200.38,E2 3200.38} C_VEL
LIN {X 0,Y 698.824,Z 762.06,A -85,B 0,C 180,E1 3207.836,E2 3207.836} C_VEL
LIN {X 0,Y 698.692,Z 762.06,A -85,B 0,C 180,E1 3214.923,E2 3214.923} C_VEL
LIN {X 0,Y 698.857,Z 762.06,A -85,B 0,C 180,E1 3222.937,E2 3222.937} C_VEL
LIN {X 0,Y 698.895,Z 762.06,A -85,B 0,C 180,E1 3230.848,E2 3230.848} C_VEL
LIN {X 0,Y 699.113,Z 762.06,A -85,B 0,C 180,E1 3238.121,E2 3238.121} C_VEL
LIN {X 0,Y 699.143,Z 762.06,A -85,B 0,C 180,E1 3245.594,E2 3245.594} C_VEL
LIN {X 0,Y 699.04,Z 762.06,A -85,B 0,C 180,E1 3253.165,E2 3253.165} C_VEL
LIN {X 0,Y 698.828,Z 762.06,A -85,B 0,C 180,E1 3260.986,E2 3260.986} C_VEL
LIN {X 0,Y 698.919,Z 762.06,A -85,B 0,C 180,E1 3269.235,E2 3269.235} C_VEL
LIN {X 0,Y 698.675,Z 762.06,A -85,B 0,C 180,E1 3276.669,E2 3276.669} C_VEL
LIN {X 0,Y 698.684,Z 762.06,A -85,B 0,C 180,E1 3283.356,E2 3283.356} C_VEL
LIN {X 0,Y 698.764,Z 762.06,A -85,B 0,C 180,E1 3292.429,E2 3292.429} C_VEL
LIN {X 0,Y 698.834,Z 763.278,A -85,B 0,C 180,E1 3293.546,E2 3293.546} C_VEL
LIN {X 0,Y 709.752,Z 787.463,A -85,B 0,C 180,E1 3294.488,E2 3294.488} C_VEL
LIN {X 0,Y 709.372,Z 873.118,A -85,B 0,C 180,E1 3295.867,E2 3295.867} C_VEL
LIN {X 0,Y 707.159,Z 943.605,A -85,B 0,C 180,E1 3298.211,E2 3298.211} C_VEL
LIN {X 0,Y 704.326,Z 1010.957,A -85,B 0,C 180,E1 3301.815,E2 3301.815} C_VEL
LIN {X 0,Y 701.749,Z 1070.991,A -85,B 0,C 180,E1 3306.558,E2 3306.558} C_VEL
LIN {X 0,Y 700.101,Z 1116.484,A -85,B 0,C 180,E1 3311.695,E2 3311.695} C_VEL
LIN {X 0,Y 699.113,Z 1148.044,A -85,B 0,C 180,E1 3316.836,E2 3316.836} C_VEL
LIN {X 0,Y 699.06,Z 1168.057,A -85,B 0,C 180,E1 3321.895,E2 3321.895} C_VEL
LIN {X 0,Y 699.14,Z 1178.296,A -85,B 0,C 180,E1 3326.893,E2 3326.893} C_VEL
LIN {X 0,Y 699.27,Z 1179.264,A -85,B 0,C 180,E1 3331.865,E2 3331.865} C_VEL
LIN {X 0,Y 699.197,Z 1167.772,A -85,B 0,C 180,E1 3338.106,E2 3338.106} C_VEL
LIN {X 0,Y 699.555,Z 1144.322,A -85,B 0,C 180,E1 3343.797,E2 3343.797} C_VEL
LIN {X 0,Y 700.602,Z 1105.682,A -85,B 0,C 180,E1 3349.605,E2 3349.605} C_VEL
LIN {X 0,Y 702.536,Z 1053.811,A -85,B 0,C 180,E1 3354.895,E2 3354.895} C_VEL
LIN {X 0,Y 705.238,Z 991.247,A -85,B 0,C 180,E1 3359.306,E2 3359.306} C_VEL
LIN {X 0,Y 707.97,Z 921.751,A -85,B 0,C 180,E1 3362.559,E2 3362.559} C_VEL
LIN {X 0,Y 709.864,Z 851.237,A -85,B 0,C 180,E1 3364.508,E2 3364.508} C_VEL
LIN {X 0,Y 707.959,Z 780.465,A -85,B 0,C 180,E1 3365.611,E2 3365.611} C_VEL
LIN {X 0,Y 699.053,Z 762.06,A -85,B 0,C 180,E1 3366.398,E2 3366.398} C_VEL
LIN {X 0,Y 698.748,Z 762.06,A -85,B 0,C 180,E1 3375.111,E2 3375.111} C_VEL
LIN {X 0,Y 698.704,Z 762.06,A -85,B 0,C 180,E1 3383.333,E2 3383.333} C_VEL
LIN {X 0,Y 698.547,Z 762.06,A -85,B 0,C 180,E1 3392.165,E2 3392.165} C_VEL
LIN {X 0,Y 698.786,Z 762.06,A -85,B 0,C 180,E1 3399.012,E2 3399.012} C_VEL
LIN {X 0,Y 699.458,Z 762.06,A -85,B 0,C 180,E1 3408.116,E2 3408.116} C_VEL
LIN {X 0,Y 699.14,Z 762.06,A -85,B 0,C 180,E1 3418.147,E2 3418.147} C_VEL
LIN {X 0,Y 699.109,Z 762.06,A -85,B 0,C 180,E1 3425.619,E2 3425.619} C_VEL
LIN {X 0,Y 699.038,Z 762.06,A -85,B 0,C 180,E1 3433.191,E2 3433.191} C_VEL
LIN {X 0,Y 698.58,Z 762.06,A -85,B 0,C 180,E1 3438.448,E2 3438.448} C_VEL
LIN {X 0,Y 690.694,Z 762.06,A -85,B 0,C 180,E1 3441.31,E2 3441.31} C_VEL
LIN {X 0,Y 690.557,Z 762.06,A -85,B 0,C 180,E1 3449.834,E2 3449.834} C_VEL
LIN {X 0,Y 690.545,Z 762.06,A -85,B 0,C 180,E1 3457.205,E2 3457.205} C_VEL
LIN {X 0,Y 690.457,Z 762.06,A -85,B 0,C 180,E1 3466.221,E2 3466.221} C_VEL
LIN {X 0,Y 690.036,Z 763.373,A -85,B 0,C 180,E1 3469.069,E2 3469.069} C_VEL
LIN {X 0,Y 705.994,Z 794.03,A -85,B 0,C 180,E1 3470.579,E2 3470.579} C_VEL
LIN {X 0,Y 704.981,Z 875.113,A -85,B 0,C 180,E1 3471.977,E2 3471.977} C_VEL
LIN {X 0,Y 702.162,Z 945.825,A -85,B 0,C 180,E1 3474.365,E2 3474.365} C_VEL
LIN {X 0,Y 698.662,Z 1015.732,A -85,B 0,C 180,E1 3478.058,E2 3478.058} C_VEL
LIN {X 0,Y 695.192,Z 1079.487,A -85,B 0,C 180,E1 3482.928,E2 3482.928} C_VEL
LIN {X 0,Y 692.79,Z 1129.724,A -85,B 0,C 180,E1 3488.305,E2 3488.305} C_VEL
LIN {X 0,Y 691.567,Z 1166.142,A -85,B 0,C 180,E1 3493.763,E2 3493.763} C_VEL
LIN {X 0,Y 691.002,Z 1192.182,A -85,B 0,C 180,E1 3499.567,E2 3499.567} C_VEL
LIN {X 0,Y 691.021,Z 1205.88,A -85,B 0,C 180,E1 3504.963,E2 3504.963} C_VEL
LIN {X 0,Y 690.869,Z 1209.727,A -85,B 0,C 180,E1 3511.038,E2 3511.038} C_VEL
LIN {X 0,Y 691.075,Z 1203.526,A -85,B 0,C 180,E1 3516.298,E2 3516.298} C_VEL
LIN {X 0,Y 691.224,Z 1185.44,A -85,B 0,C 180,E1 3522.214,E2 3522.214} C_VEL
LIN {X 0,Y 691.92,Z 1154.422,A -85,B 0,C 180,E1 3528.223,E2 3528.223} C_VEL
LIN {X 0,Y 693.855,Z 1109.44,A -85,B 0,C 180,E1 3534.087,E2 3534.087} C_VEL
LIN {X 0,Y 696.764,Z 1051.667,A -85,B 0,C 180,E1 3539.41,E2 3539.41} C_VEL
LIN {X 0,Y 700.322,Z 984.523,A -85,B 0,C 180,E1 3543.774,E2 3543.774} C_VEL
LIN {X 0,Y 703.625,Z 913.181,A -85,B 0,C 180,E1 3546.892,E2 3546.892} C_VEL
LIN {X 0,Y 705.736,Z 838.687,A -85,B 0,C 180,E1 3548.799,E2 3548.799} C_VEL
LIN {X 0,Y 704.512,Z 787.998,A -85,B 0,C 180,E1 3549.598,E2 3549.598} C_VEL
LIN {X 0,Y 691.096,Z 762.06,A -85,B 0,C 180,E1 3551.055,E2 3551.055} C_VEL
LIN {X 0,Y 690.777,Z 762.06,A -85,B 0,C 180,E1 3561.212,E2 3561.212} C_VEL
LIN {X 0,Y 690.606,Z 762.06,A -85,B 0,C 180,E1 3568.889,E2 3568.889} C_VEL
LIN {X 0,Y 690.315,Z 762.06,A -85,B 0,C 180,E1 3575.984,E2 3575.984} C_VEL
LIN {X 0,Y 690.877,Z 762.06,A -85,B 0,C 180,E1 3582.734,E2 3582.734} C_VEL
LIN {X 0,Y 690.994,Z 762.06,A -85,B 0,C 180,E1 3590.505,E2 3590.505} C_VEL
LIN {X 0,Y 691.117,Z 762.06,A -85,B 0,C 180,E1 3598.099,E2 3598.099} C_VEL
LIN {X 0,Y 691.112,Z 762.06,A -85,B 0,C 180,E1 3605.659,E2 3605.659} C_VEL
LIN {X 0,Y 690.942,Z 762.06,A -85,B 0,C 180,E1 3613.322,E2 3613.322} C_VEL
LIN {X 0,Y 690.7,Z 762.06,A -85,B 0,C 180,E1 3621.245,E2 3621.245} C_VEL
LIN {X 0,Y 690.767,Z 762.06,A -85,B 0,C 180,E1 3629.87,E2 3629.87} C_VEL
LIN {X 0,Y 690.547,Z 762.06,A -85,B 0,C 180,E1 3637.172,E2 3637.172} C_VEL
LIN {X 0,Y 690.339,Z 762.06,A -85,B 0,C 180,E1 3644.445,E2 3644.445} C_VEL
LIN {X 0,Y 690.733,Z 762.06,A -85,B 0,C 180,E1 3652.983,E2 3652.983} C_VEL
LIN {X 0,Y 703.221,Z 790.964,A -85,B 0,C 180,E1 3654.151,E2 3654.151} C_VEL
LIN {X 0,Y 702.65,Z 875.344,A -85,B 0,C 180,E1 3655.554,E2 3655.554} C_VEL
LIN {X 0,Y 700.123,Z 945.675,A -85,B 0,C 180,E1 3657.95,E2 3657.95} C_VEL
LIN {X 0,Y 696.925,Z 1013.315,A -85,B 0,C 180,E1 3661.654,E2 3661.654} C_VEL
LIN {X 0,Y 694.085,Z 1071.616,A -85,B 0,C 180,E1 3666.345,E2 3666.345} C_VEL
LIN {X 0,Y 692.24,Z 1117.519,A -85,B 0,C 180,E1 3671.623,E2 3671.623} C_VEL
LIN {X 0,Y 691.131,Z 1149.553,A -85,B 0,C 180,E1 3676.995,E2 3676.995} C_VEL
LIN {X 0,Y 690.939,Z 1169.893,A -85,B 0,C 180,E1 3682.434,E2 3682.434} C_VEL
LIN {X 0,Y 691.148,Z 1178.295,A -85,B 0,C 180,E1 3686.857,E2 3686.857} C_VEL
LIN {X 0,Y 691.118,Z 1178.744,A -85,B 0,C 180,E1 3692.53,E2 3692.53} C_VEL
LIN {X 0,Y 691.179,Z 1167.774,A -85,B 0,C 180,E1 3698.201,E2 3698.201} C_VEL
LIN {X 0,Y 691.588,Z 1144.323,A -85,B 0,C 180,E1 3703.959,E2 3703.959} C_VEL
LIN {X 0,Y 692.82,Z 1105.688,A -85,B 0,C 180,E1 3709.834,E2 3709.834} C_VEL
LIN {X 0,Y 694.948,Z 1053.817,A -85,B 0,C 180,E1 3715.185,E2 3715.185} C_VEL
LIN {X 0,Y 698.1,Z 991.261,A -85,B 0,C 180,E1 3719.635,E2 3719.635} C_VEL
LIN {X 0,Y 701.098,Z 922.779,A -85,B 0,C 180,E1 3722.88,E2 3722.88} C_VEL
LIN {X 0,Y 703.243,Z 852.639,A -85,B 0,C 180,E1 3724.854,E2 3724.854} C_VEL
LIN {X 0,Y 701.606,Z 783.591,A -85,B 0,C 180,E1 3725.945,E2 3725.945} C_VEL
LIN {X 0,Y 690.842,Z 762.06,A -85,B 0,C 180,E1 3726.95,E2 3726.95} C_VEL
LIN {X 0,Y 690.546,Z 762.06,A -85,B 0,C 180,E1 3736.2,E2 3736.2} C_VEL
LIN {X 0,Y 690.485,Z 762.06,A -85,B 0,C 180,E1 3744.388,E2 3744.388} C_VEL
LIN {X 0,Y 690.61,Z 762.06,A -85,B 0,C 180,E1 3751.817,E2 3751.817} C_VEL
LIN {X 0,Y 690.477,Z 762.06,A -85,B 0,C 180,E1 3760.093,E2 3760.093} C_VEL
LIN {X 0,Y 691.43,Z 762.06,A -85,B 0,C 180,E1 3767.976,E2 3767.976} C_VEL
LIN {X 0,Y 691.144,Z 762.06,A -85,B 0,C 180,E1 3778.125,E2 3778.125} C_VEL
LIN {X 0,Y 691.089,Z 762.06,A -85,B 0,C 180,E1 3785.685,E2 3785.685} C_VEL
LIN {X 0,Y 690.951,Z 762.06,A -85,B 0,C 180,E1 3793.349,E2 3793.349} C_VEL
LIN {X 0,Y 690.694,Z 762.06,A -85,B 0,C 180,E1 3801.31,E2 3801.31} C_VEL
LIN {X 0,Y 681.966,Z 762.06,A -85,B 0,C 180,E1 3804.183,E2 3804.183} C_VEL
LIN {X 0,Y 682.216,Z 762.06,A -85,B 0,C 180,E1 3811.147,E2 3811.147} C_VEL
LIN {X 0,Y 682.3,Z 762.06,A -85,B 0,C 180,E1 3817.902,E2 3817.902} C_VEL
LIN {X 0,Y 682.423,Z 762.06,A -85,B 0,C 180,E1 3826.309,E2 3826.309} C_VEL
LIN {X 0,Y 682.096,Z 763.464,A -85,B 0,C 180,E1 3828.489,E2 3828.489} C_VEL
LIN {X 0,Y 699.816,Z 795.884,A -85,B 0,C 180,E1 3830.186,E2 3830.186} C_VEL
LIN {X 0,Y 698.618,Z 875.115,A -85,B 0,C 180,E1 3831.568,E2 3831.568} C_VEL
LIN {X 0,Y 695.488,Z 945.829,A -85,B 0,C 180,E1 3833.97,E2 3833.97} C_VEL
LIN {X 0,Y 691.569,Z 1015.758,A -85,B 0,C 180,E1 3837.693,E2 3837.693} C_VEL
LIN {X 0,Y 687.705,Z 1080.083,A -85,B 0,C 180,E1 3842.664,E2 3842.664} C_VEL
LIN {X 0,Y 684.984,Z 1131.169,A -85,B 0,C 180,E1 3848.232,E2 3848.232} C_VEL
LIN {X 0,Y 683.555,Z 1167.908,A -85,B 0,C 180,E1 3853.898,E2 3853.898} C_VEL
LIN {X 0,Y 682.96,Z 1193.293,A -85,B 0,C 180,E1 3859.766,E2 3859.766} C_VEL
LIN {X 0,Y 682.822,Z 1206.827,A -85,B 0,C 180,E1 3865.54,E2 3865.54} C_VEL
LIN {X 0,Y 683.016,Z 1209.838,A -85,B 0,C 180,E1 3870.635,E2 3870.635} C_VEL
LIN {X 0,Y 683.04,Z 1203.526,A -85,B 0,C 180,E1 3876.372,E2 3876.372} C_VEL
LIN {X 0,Y 683.202,Z 1185.44,A -85,B 0,C 180,E1 3882.36,E2 3882.36} C_VEL
LIN {X 0,Y 684.056,Z 1156.562,A -85,B 0,C 180,E1 3888.08,E2 3888.08} C_VEL
LIN {X 0,Y 686.087,Z 1112.517,A -85,B 0,C 180,E1 3894.017,E2 3894.017} C_VEL
LIN {X 0,Y 689.184,Z 1056.213,A -85,B 0,C 180,E1 3899.393,E2 3899.393} C_VEL
LIN {X 0,Y 693.201,Z 989.176,A -85,B 0,C 180,E1 3903.907,E2 3903.907} C_VEL
LIN {X 0,Y 696.859,Z 918.097,A -85,B 0,C 180,E1 3907.122,E2 3907.122} C_VEL
LIN {X 0,Y 699.309,Z 843.631,A -85,B 0,C 180,E1 3909.125,E2 3909.125} C_VEL
LIN {X 0,Y 698.362,Z 791.344,A -85,B 0,C 180,E1 3909.973,E2 3909.973} C_VEL
LIN {X 0,Y 683.023,Z 762.06,A -85,B 0,C 180,E1 3911.577,E2 3911.577} C_VEL
LIN {X 0,Y 682.701,Z 762.06,A -85,B 0,C 180,E1 3920.665,E2 3920.665} C_VEL
LIN {X 0,Y 682.617,Z 762.06,A -85,B 0,C 180,E1 3928.793,E2 3928.793} C_VEL
LIN {X 0,Y 682.43,Z 762.06,A -85,B 0,C 180,E1 3935.689,E2 3935.689} C_VEL
LIN {X 0,Y 682.502,Z 762.06,A -85,B 0,C 180,E1 3943.846,E2 3943.846} C_VEL
LIN {X 0,Y 682.56,Z 762.06,A -85,B 0,C 180,E1 3951.676,E2 3951.676} C_VEL
LIN {X 0,Y 683.125,Z 762.06,A -85,B 0,C 180,E1 3958.077,E2 3958.077} C_VEL
LIN {X 0,Y 683.062,Z 762.06,A -85,B 0,C 180,E1 3965.726,E2 3965.726} C_VEL
LIN {X 0,Y 682.851,Z 762.06,A -85,B 0,C 180,E1 3973.483,E2 3973.483} C_VEL
LIN {X 0,Y 682.573,Z 762.06,A -85,B 0,C 180,E1 3981.511,E2 3981.511} C_VEL
LIN {X 0,Y 682.764,Z 762.06,A -85,B 0,C 180,E1 3989.997,E2 3989.997} C_VEL
LIN {X 0,Y 682.413,Z 762.06,A -85,B 0,C 180,E1 3997.918,E2 3997.918} C_VEL
LIN {X 0,Y 682.141,Z 762.06,A -85,B 0,C 180,E1 4005.551,E2 4005.551} C_VEL
LIN {X 0,Y 682.881,Z 763.638,A -85,B 0,C 180,E1 4012.557,E2 4012.557} C_VEL
LIN {X 0,Y 696.758,Z 793.876,A -85,B 0,C 180,E1 4013.804,E2 4013.804} C_VEL
LIN {X 0,Y 695.952,Z 876.58,A -85,B 0,C 180,E1 4015.211,E2 4015.211} C_VEL
LIN {X 0,Y 693.189,Z 945.658,A -85,B 0,C 180,E1 4017.59,E2 4017.59} C_VEL
LIN {X 0,Y 689.638,Z 1013.185,A -85,B 0,C 180,E1 4021.319,E2 4021.319} C_VEL
LIN {X 0,Y 686.411,Z 1072.914,A -85,B 0,C 180,E1 4026.192,E2 4026.192} C_VEL
LIN {X 0,Y 684.342,Z 1118.885,A -85,B 0,C 180,E1 4031.593,E2 4031.593} C_VEL
LIN {X 0,Y 683.184,Z 1149.593,A -85,B 0,C 180,E1 4036.85,E2 4036.85} C_VEL
LIN {X 0,Y 682.983,Z 1169.892,A -85,B 0,C 180,E1 4042.345,E2 4042.345} C_VEL
LIN {X 0,Y 683.155,Z 1178.295,A -85,B 0,C 180,E1 4046.82,E2 4046.82} C_VEL
LIN {X 0,Y 683.267,Z 1179.265,A -85,B 0,C 180,E1 4051.909,E2 4051.909} C_VEL
LIN {X 0,Y 683.441,Z 1169.664,A -85,B 0,C 180,E1 4057.652,E2 4057.652} C_VEL
LIN {X 0,Y 683.676,Z 1146.049,A -85,B 0,C 180,E1 4063.797,E2 4063.797} C_VEL
LIN {X 0,Y 684.957,Z 1107.658,A -85,B 0,C 180,E1 4069.822,E2 4069.822} C_VEL
LIN {X 0,Y 687.325,Z 1055.735,A -85,B 0,C 180,E1 4075.311,E2 4075.311} C_VEL
LIN {X 0,Y 690.774,Z 994.094,A -85,B 0,C 180,E1 4079.809,E2 4079.809} C_VEL
LIN {X 0,Y 694.201,Z 925.355,A -85,B 0,C 180,E1 4083.149,E2 4083.149} C_VEL
LIN {X 0,Y 696.625,Z 854.279,A -85,B 0,C 180,E1 4085.202,E2 4085.202} C_VEL
LIN {X 0,Y 695.306,Z 786.711,A -85,B 0,C 180,E1 4086.284,E2 4086.284} C_VEL
LIN {X 0,Y 682.627,Z 762.06,A -85,B 0,C 180,E1 4087.487,E2 4087.487} C_VEL
LIN {X 0,Y 682.534,Z 762.06,A -85,B 0,C 180,E1 4096.231,E2 4096.231} C_VEL
LIN {X 0,Y 682.509,Z 762.06,A -85,B 0,C 180,E1 4104.198,E2 4104.198} C_VEL
LIN {X 0,Y 682.614,Z 762.06,A -85,B 0,C 180,E1 4111.456,E2 4111.456} C_VEL
LIN {X 0,Y 682.519,Z 762.06,A -85,B 0,C 180,E1 4119.851,E2 4119.851} C_VEL
LIN {X 0,Y 683.434,Z 762.06,A -85,B 0,C 180,E1 4127.834,E2 4127.834} C_VEL
LIN {X 0,Y 683.152,Z 762.06,A -85,B 0,C 180,E1 4138.103,E2 4138.103} C_VEL
LIN {X 0,Y 683.04,Z 762.06,A -85,B 0,C 180,E1 4145.752,E2 4145.752} C_VEL
LIN {X 0,Y 682.86,Z 762.06,A -85,B 0,C 180,E1 4153.51,E2 4153.51} C_VEL
LIN {X 0,Y 682.584,Z 762.06,A -85,B 0,C 180,E1 4161.538,E2 4161.538} C_VEL
LIN {X 0,Y 681.966,Z 762.06,A -85,B 0,C 180,E1 4164.183,E2 4164.183} C_VEL
LIN {X 0,Y 674.498,Z 762.06,A -85,B 0,C 180,E1 4167.121,E2 4167.121} C_VEL
LIN {X 0,Y 674.347,Z 762.06,A -85,B 0,C 180,E1 4175.042,E2 4175.042} C_VEL
LIN {X 0,Y 674.537,Z 762.06,A -85,B 0,C 180,E1 4184.91,E2 4184.91} C_VEL
LIN {X 0,Y 674.102,Z 762.558,A -85,B 0,C 180,E1 4187.872,E2 4187.872} C_VEL
LIN {X 0,Y 693.628,Z 801.607,A -85,B 0,C 180,E1 4189.835,E2 4189.835} C_VEL
LIN {X 0,Y 692.139,Z 879.341,A -85,B 0,C 180,E1 4191.264,E2 4191.264} C_VEL
LIN {X 0,Y 688.696,Z 949.26,A -85,B 0,C 180,E1 4193.716,E2 4193.716} C_VEL
LIN {X 0,Y 684.302,Z 1019.61,A -85,B 0,C 180,E1 4197.57,E2 4197.57} C_VEL
LIN {X 0,Y 680.138,Z 1082.215,A -85,B 0,C 180,E1 4202.534,E2 4202.534} C_VEL
LIN {X 0,Y 677.169,Z 1132.495,A -85,B 0,C 180,E1 4208.14,E2 4208.14} C_VEL
LIN {X 0,Y 675.682,Z 1167.91,A -85,B 0,C 180,E1 4213.706,E2 4213.706} C_VEL
LIN {X 0,Y 675.026,Z 1193.293,A -85,B 0,C 180,E1 4219.645,E2 4219.645} C_VEL
LIN {X 0,Y 674.836,Z 1206.824,A -85,B 0,C 180,E1 4225.488,E2 4225.488} C_VEL
LIN {X 0,Y 675.02,Z 1209.838,A -85,B 0,C 180,E1 4230.642,E2 4230.642} C_VEL
LIN {X 0,Y 675.027,Z 1203.526,A -85,B 0,C 180,E1 4236.448,E2 4236.448} C_VEL
LIN {X 0,Y 675.255,Z 1186.211,A -85,B 0,C 180,E1 4242.318,E2 4242.318} C_VEL
LIN {X 0,Y 676.107,Z 1156.564,A -85,B 0,C 180,E1 4248.3,E2 4248.3} C_VEL
LIN {X 0,Y 678.396,Z 1113.281,A -85,B 0,C 180,E1 4254.216,E2 4254.216} C_VEL
LIN {X 0,Y 681.92,Z 1056.212,A -85,B 0,C 180,E1 4259.738,E2 4259.738} C_VEL
LIN {X 0,Y 686.334,Z 989.174,A -85,B 0,C 180,E1 4264.293,E2 4264.293} C_VEL
LIN {X 0,Y 690.391,Z 918.094,A -85,B 0,C 180,E1 4267.529,E2 4267.529} C_VEL
LIN {X 0,Y 693.131,Z 842.955,A -85,B 0,C 180,E1 4269.555,E2 4269.555} C_VEL
LIN {X 0,Y 692.426,Z 794.863,A -85,B 0,C 180,E1 4270.339,E2 4270.339} C_VEL
LIN {X 0,Y 674.908,Z 762.06,A -85,B 0,C 180,E1 4272.184,E2 4272.184} C_VEL
LIN {X 0,Y 674.673,Z 762.06,A -85,B 0,C 180,E1 4281.765,E2 4281.765} C_VEL
LIN {X 0,Y 674.496,Z 762.06,A -85,B 0,C 180,E1 4289.951,E2 4289.951} C_VEL
LIN {X 0,Y 674.107,Z 762.06,A -85,B 0,C 180,E1 4296.78,E2 4296.78} C_VEL
LIN {X 0,Y 674.535,Z 762.06,A -85,B 0,C 180,E1 4303.65,E2 4303.65} C_VEL
LIN {X 0,Y 674.598,Z 762.06,A -85,B 0,C 180,E1 4311.577,E2 4311.577} C_VEL
LIN {X 0,Y 675.135,Z 762.06,A -85,B 0,C 180,E1 4318.054,E2 4318.054} C_VEL
LIN {X 0,Y 675.042,Z 762.06,A -85,B 0,C 180,E1 4325.794,E2 4325.794} C_VEL
LIN {X 0,Y 674.767,Z 762.06,A -85,B 0,C 180,E1 4333.648,E2 4333.648} C_VEL
LIN {X 0,Y 674.458,Z 762.06,A -85,B 0,C 180,E1 4341.783,E2 4341.783} C_VEL
LIN {X 0,Y 674.723,Z 762.06,A -85,B 0,C 180,E1 4350.392,E2 4350.392} C_VEL
LIN {X 0,Y 674.4,Z 762.06,A -85,B 0,C 180,E1 4358.22,E2 4358.22} C_VEL
LIN {X 0,Y 674.203,Z 762.06,A -85,B 0,C 180,E1 4365.147,E2 4365.147} C_VEL
LIN {X 0,Y 674.984,Z 763.925,A -85,B 0,C 180,E1 4372.047,E2 4372.047} C_VEL
LIN {X 0,Y 690.313,Z 794.873,A -85,B 0,C 180,E1 4373.424,E2 4373.424} C_VEL
LIN {X 0,Y 689.256,Z 878.12,A -85,B 0,C 180,E1 4374.87,E2 4374.87} C_VEL
LIN {X 0,Y 686.175,Z 947.761,A -85,B 0,C 180,E1 4377.322,E2 4377.322} C_VEL
LIN {X 0,Y 682.294,Z 1014.724,A -85,B 0,C 180,E1 4381.092,E2 4381.092} C_VEL
LIN {X 0,Y 678.824,Z 1073.335,A -85,B 0,C 180,E1 4385.952,E2 4385.952} C_VEL
LIN {X 0,Y 676.51,Z 1118.879,A -85,B 0,C 180,E1 4391.372,E2 4391.372} C_VEL
LIN {X 0,Y 675.261,Z 1149.591,A -85,B 0,C 180,E1 4396.693,E2 4396.693} C_VEL
LIN {X 0,Y 675.016,Z 1169.891,A -85,B 0,C 180,E1 4402.254,E2 4402.254} C_VEL
LIN {X 0,Y 675.165,Z 1178.294,A -85,B 0,C 180,E1 4406.782,E2 4406.782} C_VEL
LIN {X 0,Y 675.282,Z 1179.265,A -85,B 0,C 180,E1 4411.932,E2 4411.932} C_VEL
LIN {X 0,Y 675.415,Z 1169.666,A -85,B 0,C 180,E1 4417.744,E2 4417.744} C_VEL
LIN {X 0,Y 675.693,Z 1146.052,A -85,B 0,C 180,E1 4423.963,E2 4423.963} C_VEL
LIN {X 0,Y 677.171,Z 1107.659,A -85,B 0,C 180,E1 4430.06,E2 4430.06} C_VEL
LIN {X 0,Y 679.72,Z 1057.301,A -85,B 0,C 180,E1 4435.47,E2 4435.47} C_VEL
LIN {X 0,Y 683.522,Z 995.687,A -85,B 0,C 180,E1 4440.053,E2 4440.053} C_VEL
LIN {X 0,Y 687.283,Z 928.168,A -85,B 0,C 180,E1 4443.412,E2 4443.412} C_VEL
LIN {X 0,Y 689.958,Z 857.836,A -85,B 0,C 180,E1 4445.515,E2 4445.515} C_VEL
LIN {X 0,Y 688.968,Z 789.96,A -85,B 0,C 180,E1 4446.631,E2 4446.631} C_VEL
LIN {X 0,Y 674.456,Z 762.06,A -85,B 0,C 180,E1 4447.949,E2 4447.949} C_VEL
LIN {X 0,Y 674.383,Z 762.06,A -85,B 0,C 180,E1 4456.959,E2 4456.959} C_VEL
LIN {X 0,Y 674.293,Z 762.06,A -85,B 0,C 180,E1 4465.177,E2 4465.177} C_VEL
LIN {X 0,Y 674.396,Z 762.06,A -85,B 0,C 180,E1 4472.655,E2 4472.655} C_VEL
LIN {X 0,Y 674.541,Z 762.06,A -85,B 0,C 180,E1 4479.602,E2 4479.602} C_VEL
LIN {X 0,Y 675.416,Z 762.06,A -85,B 0,C 180,E1 4487.687,E2 4487.687} C_VEL
LIN {X 0,Y 675.157,Z 762.06,A -85,B 0,C 180,E1 4498.081,E2 4498.081} C_VEL
LIN {X 0,Y 675.005,Z 762.06,A -85,B 0,C 180,E1 4505.821,E2 4505.821} C_VEL
LIN {X 0,Y 674.774,Z 762.06,A -85,B 0,C 180,E1 4513.675,E2 4513.675} C_VEL
LIN {X 0,Y 674.478,Z 762.06,A -85,B 0,C 180,E1 4521.81,E2 4521.81} C_VEL
LIN {X 0,Y 674.498,Z 762.06,A -85,B 0,C 180,E1 4527.121,E2 4527.121} C_VEL
LIN {X 0,Y 666.362,Z 762.06,A -85,B 0,C 180,E1 4530.089,E2 4530.089} C_VEL
LIN {X 0,Y 666.046,Z 762.06,A -85,B 0,C 180,E1 4538.823,E2 4538.823} C_VEL
LIN {X 0,Y 666.207,Z 762.486,A -85,B 0,C 180,E1 4547.254,E2 4547.254} C_VEL
LIN {X 0,Y 687.483,Z 804.116,A -85,B 0,C 180,E1 4549.435,E2 4549.435} C_VEL
LIN {X 0,Y 685.676,Z 882.394,A -85,B 0,C 180,E1 4550.924,E2 4550.924} C_VEL
LIN {X 0,Y 681.837,Z 953.409,A -85,B 0,C 180,E1 4553.49,E2 4553.49} C_VEL
LIN {X 0,Y 676.974,Z 1023.79,A -85,B 0,C 180,E1 4557.47,E2 4557.47} C_VEL
LIN {X 0,Y 672.423,Z 1085.946,A -85,B 0,C 180,E1 4562.569,E2 4562.569} C_VEL
LIN {X 0,Y 669.132,Z 1136.292,A -85,B 0,C 180,E1 4568.397,E2 4568.397} C_VEL
LIN {X 0,Y 667.563,Z 1171.414,A -85,B 0,C 180,E1 4574.179,E2 4574.179} C_VEL
LIN {X 0,Y 666.992,Z 1194.316,A -85,B 0,C 180,E1 4579.85,E2 4579.85} C_VEL
LIN {X 0,Y 666.851,Z 1206.821,A -85,B 0,C 180,E1 4585.433,E2 4585.433} C_VEL
LIN {X 0,Y 667.015,Z 1209.838,A -85,B 0,C 180,E1 4590.65,E2 4590.65} C_VEL
LIN {X 0,Y 667.006,Z 1203.526,A -85,B 0,C 180,E1 4596.526,E2 4596.526} C_VEL
LIN {X 0,Y 667.247,Z 1186.21,A -85,B 0,C 180,E1 4602.468,E2 4602.468} C_VEL
LIN {X 0,Y 668.196,Z 1156.565,A -85,B 0,C 180,E1 4608.525,E2 4608.525} C_VEL
LIN {X 0,Y 670.689,Z 1112.899,A -85,B 0,C 180,E1 4614.558,E2 4614.558} C_VEL
LIN {X 0,Y 674.622,Z 1056.379,A -85,B 0,C 180,E1 4620.077,E2 4620.077} C_VEL
LIN {X 0,Y 679.51,Z 989.171,A -85,B 0,C 180,E1 4624.686,E2 4624.686} C_VEL
LIN {X 0,Y 683.985,Z 917.367,A -85,B 0,C 180,E1 4627.973,E2 4627.973} C_VEL
LIN {X 0,Y 686.921,Z 843.807,A -85,B 0,C 180,E1 4629.966,E2 4629.966} C_VEL
LIN {X 0,Y 686.169,Z 797.712,A -85,B 0,C 180,E1 4630.746,E2 4630.746} C_VEL
LIN {X 0,Y 666.791,Z 762.06,A -85,B 0,C 180,E1 4632.746,E2 4632.746} C_VEL
LIN {X 0,Y 666.683,Z 762.06,A -85,B 0,C 180,E1 4641.698,E2 4641.698} C_VEL
LIN {X 0,Y 666.508,Z 762.06,A -85,B 0,C 180,E1 4649.162,E2 4649.162} C_VEL
LIN {X 0,Y 666.179,Z 762.06,A -85,B 0,C 180,E1 4656.488,E2 4656.488} C_VEL
LIN {X 0,Y 666.603,Z 762.06,A -85,B 0,C 180,E1 4663.45,E2 4663.45} C_VEL
LIN {X 0,Y 666.568,Z 762.06,A -85,B 0,C 180,E1 4671.749,E2 4671.749} C_VEL
LIN {X 0,Y 667.138,Z 762.06,A -85,B 0,C 180,E1 4678.031,E2 4678.031} C_VEL
LIN {X 0,Y 666.993,Z 762.06,A -85,B 0,C 180,E1 4685.864,E2 4685.864} C_VEL
LIN {X 0,Y 666.69,Z 762.06,A -85,B 0,C 180,E1 4693.816,E2 4693.816} C_VEL
LIN {X 0,Y 666.342,Z 762.06,A -85,B 0,C 180,E1 4702.062,E2 4702.062} C_VEL
LIN {X 0,Y 666.64,Z 762.06,A -85,B 0,C 180,E1 4710.8,E2 4710.8} C_VEL
LIN {X 0,Y 666.361,Z 762.06,A -85,B 0,C 180,E1 4718.766,E2 4718.766} C_VEL
LIN {X 0,Y 666.101,Z 762.06,A -85,B 0,C 180,E1 4726.023,E2 4726.023} C_VEL
LIN {X 0,Y 666.783,Z 762.738,A -85,B 0,C 180,E1 4731.48,E2 4731.48} C_VEL
LIN {X 0,Y 683.864,Z 797.668,A -85,B 0,C 180,E1 4733.059,E2 4733.059} C_VEL
LIN {X 0,Y 682.588,Z 879.709,A -85,B 0,C 180,E1 4734.523,E2 4734.523} C_VEL
LIN {X 0,Y 679.212,Z 949.223,A -85,B 0,C 180,E1 4737.018,E2 4737.018} C_VEL
LIN {X 0,Y 674.861,Z 1017.4,A -85,B 0,C 180,E1 4740.938,E2 4740.938} C_VEL
LIN {X 0,Y 671.089,Z 1075.738,A -85,B 0,C 180,E1 4745.9,E2 4745.9} C_VEL
LIN {X 0,Y 668.586,Z 1121.187,A -85,B 0,C 180,E1 4751.486,E2 4751.486} C_VEL
LIN {X 0,Y 667.262,Z 1151.131,A -85,B 0,C 180,E1 4756.865,E2 4756.865} C_VEL
LIN {X 0,Y 667.039,Z 1170.038,A -85,B 0,C 180,E1 4762.223,E2 4762.223} C_VEL
LIN {X 0,Y 667.171,Z 1178.294,A -85,B 0,C 180,E1 4766.744,E2 4766.744} C_VEL
LIN {X 0,Y 667.272,Z 1179.266,A -85,B 0,C 180,E1 4771.955,E2 4771.955} C_VEL
LIN {X 0,Y 667.181,Z 1168.177,A -85,B 0,C 180,E1 4778.362,E2 4778.362} C_VEL
LIN {X 0,Y 667.692,Z 1144.721,A -85,B 0,C 180,E1 4784.393,E2 4784.393} C_VEL
LIN {X 0,Y 669.331,Z 1107.41,A -85,B 0,C 180,E1 4790.338,E2 4790.338} C_VEL
LIN {X 0,Y 672.251,Z 1057.303,A -85,B 0,C 180,E1 4795.774,E2 4795.774} C_VEL
LIN {X 0,Y 676.39,Z 995.97,A -85,B 0,C 180,E1 4800.385,E2 4800.385} C_VEL
LIN {X 0,Y 680.438,Z 928.845,A -85,B 0,C 180,E1 4803.764,E2 4803.764} C_VEL
LIN {X 0,Y 683.456,Z 857.536,A -85,B 0,C 180,E1 4805.913,E2 4805.913} C_VEL
LIN {X 0,Y 682.425,Z 792.653,A -85,B 0,C 180,E1 4807.006,E2 4807.006} C_VEL
LIN {X 0,Y 666.273,Z 762.06,A -85,B 0,C 180,E1 4808.513,E2 4808.513} C_VEL
LIN {X 0,Y 666.442,Z 762.06,A -85,B 0,C 180,E1 4816.021,E2 4816.021} C_VEL
LIN {X 0,Y 666.344,Z 762.06,A -85,B 0,C 180,E1 4824.507,E2 4824.507} C_VEL
LIN {X 0,Y 666.418,Z 762.06,A -85,B 0,C 180,E1 4832.182,E2 4832.182} C_VEL
LIN {X 0,Y 666.602,Z 762.06,A -85,B 0,C 180,E1 4839.348,E2 4839.348} C_VEL
LIN {X 0,Y 667.408,Z 762.06,A -85,B 0,C 180,E1 4847.537,E2 4847.537} C_VEL
LIN {X 0,Y 667.16,Z 762.06,A -85,B 0,C 180,E1 4858.058,E2 4858.058} C_VEL
LIN {X 0,Y 666.956,Z 762.06,A -85,B 0,C 180,E1 4865.891,E2 4865.891} C_VEL
LIN {X 0,Y 666.691,Z 762.06,A -85,B 0,C 180,E1 4873.844,E2 4873.844} C_VEL
LIN {X 0,Y 666.366,Z 762.06,A -85,B 0,C 180,E1 4882.09,E2 4882.09} C_VEL
LIN {X 0,Y 666.362,Z 762.06,A -85,B 0,C 180,E1 4890.089,E2 4890.089} C_VEL
LIN {X 0,Y 658.024,Z 762.06,A -85,B 0,C 180,E1 4893.066,E2 4893.066} C_VEL
LIN {X 0,Y 657.9,Z 762.06,A -85,B 0,C 180,E1 4899.446,E2 4899.446} C_VEL
LIN {X 0,Y 658.574,Z 763.933,A -85,B 0,C 180,E1 4906.658,E2 4906.658} C_VEL
LIN {X 0,Y 681.351,Z 807.442,A -85,B 0,C 180,E1 4909.038,E2 4909.038} C_VEL
LIN {X 0,Y 679.161,Z 886.639,A -85,B 0,C 180,E1 4910.61,E2 4910.61} C_VEL
LIN {X 0,Y 674.89,Z 958.07,A -85,B 0,C 180,E1 4913.298,E2 4913.298} C_VEL
LIN {X 0,Y 669.724,Z 1026.936,A -85,B 0,C 180,E1 4917.314,E2 4917.314} C_VEL
LIN {X 0,Y 664.764,Z 1088.436,A -85,B 0,C 180,E1 4922.486,E2 4922.486} C_VEL
LIN {X 0,Y 661.438,Z 1136.407,A -85,B 0,C 180,E1 4928.149,E2 4928.149} C_VEL
LIN {X 0,Y 659.683,Z 1171.412,A -85,B 0,C 180,E1 4933.985,E2 4933.985} C_VEL
LIN {X 0,Y 659.03,Z 1194.316,A -85,B 0,C 180,E1 4939.726,E2 4939.726} C_VEL
LIN {X 0,Y 658.869,Z 1206.818,A -85,B 0,C 180,E1 4945.378,E2 4945.378} C_VEL
LIN {X 0,Y 659.013,Z 1209.838,A -85,B 0,C 180,E1 4950.658,E2 4950.658} C_VEL
LIN {X 0,Y 658.993,Z 1203.526,A -85,B 0,C 180,E1 4956.606,E2 4956.606} C_VEL
LIN {X 0,Y 659.267,Z 1186.209,A -85,B 0,C 180,E1 4962.621,E2 4962.621} C_VEL
LIN {X 0,Y 660.32,Z 1156.567,A -85,B 0,C 180,E1 4968.754,E2 4968.754} C_VEL
LIN {X 0,Y 662.988,Z 1114.464,A -85,B 0,C 180,E1 4974.672,E2 4974.672} C_VEL
LIN {X 0,Y 667.226,Z 1058.054,A -85,B 0,C 180,E1 4980.296,E2 4980.296} C_VEL
LIN {X 0,Y 672.392,Z 992.772,A -85,B 0,C 180,E1 4984.876,E2 4984.876} C_VEL
LIN {X 0,Y 677.285,Z 921.619,A -85,B 0,C 180,E1 4988.238,E2 4988.238} C_VEL
LIN {X 0,Y 680.699,Z 845.797,A -85,B 0,C 180,E1 4990.364,E2 4990.364} C_VEL
LIN {X 0,Y 679.909,Z 800.71,A -85,B 0,C 180,E1 4991.161,E2 4991.161} C_VEL
LIN {X 0,Y 658.591,Z 762.06,A -85,B 0,C 180,E1 4993.432,E2 4993.432} C_VEL
LIN {X 0,Y 658.639,Z 762.06,A -85,B 0,C 180,E1 5002.593,E2 5002.593} C_VEL
LIN {X 0,Y 658.448,Z 762.06,A -85,B 0,C 180,E1 5010.275,E2 5010.275} C_VEL
LIN {X 0,Y 658.06,Z 762.06,A -85,B 0,C 180,E1 5017.616,E2 5017.616} C_VEL
LIN {X 0,Y 658.309,Z 762.06,A -85,B 0,C 180,E1 5024.61,E2 5024.61} C_VEL
LIN {X 0,Y 658.647,Z 762.06,A -85,B 0,C 180,E1 5031.372,E2 5031.372} C_VEL
LIN {X 0,Y 659.148,Z 762.06,A -85,B 0,C 180,E1 5038.007,E2 5038.007} C_VEL
LIN {X 0,Y 658.945,Z 762.06,A -85,B 0,C 180,E1 5045.936,E2 5045.936} C_VEL
LIN {X 0,Y 658.639,Z 762.06,A -85,B 0,C 180,E1 5053.989,E2 5053.989} C_VEL
LIN {X 0,Y 658.252,Z 762.06,A -85,B 0,C 180,E1 5062.347,E2 5062.347} C_VEL
LIN {X 0,Y 658.623,Z 762.06,A -85,B 0,C 180,E1 5071.217,E2 5071.217} C_VEL
LIN {X 0,Y 658.363,Z 762.06,A -85,B 0,C 180,E1 5079.499,E2 5079.499} C_VEL
LIN {X 0,Y 658.146,Z 762.06,A -85,B 0,C 180,E1 5087.178,E2 5087.178} C_VEL
LIN {X 0,Y 658.88,Z 763.838,A -85,B 0,C 180,E1 5090.924,E2 5090.924} C_VEL
LIN {X 0,Y 677.475,Z 802.428,A -85,B 0,C 180,E1 5092.715,E2 5092.715} C_VEL
LIN {X 0,Y 675.941,Z 881.948,A -85,B 0,C 180,E1 5094.188,E2 5094.188} C_VEL
LIN {X 0,Y 672.15,Z 952.169,A -85,B 0,C 180,E1 5096.777,E2 5096.777} C_VEL
LIN {X 0,Y 667.482,Z 1019.751,A -85,B 0,C 180,E1 5100.761,E2 5100.761} C_VEL
LIN {X 0,Y 663.451,Z 1076.684,A -85,B 0,C 180,E1 5105.706,E2 5105.706} C_VEL
LIN {X 0,Y 660.688,Z 1122.286,A -85,B 0,C 180,E1 5111.43,E2 5111.43} C_VEL
LIN {X 0,Y 659.272,Z 1152.666,A -85,B 0,C 180,E1 5117.041,E2 5117.041} C_VEL
LIN {X 0,Y 658.935,Z 1171.456,A -85,B 0,C 180,E1 5122.729,E2 5122.729} C_VEL
LIN {X 0,Y 658.767,Z 1179.339,A -85,B 0,C 180,E1 5128.022,E2 5128.022} C_VEL
LIN {X 0,Y 659.004,Z 1178.174,A -85,B 0,C 180,E1 5133.299,E2 5133.299} C_VEL
LIN {X 0,Y 659.122,Z 1167.781,A -85,B 0,C 180,E1 5138.602,E2 5138.602} C_VEL
LIN {X 0,Y 659.72,Z 1144.998,A -85,B 0,C 180,E1 5144.517,E2 5144.517} C_VEL
LIN {X 0,Y 661.494,Z 1108.695,A -85,B 0,C 180,E1 5150.421,E2 5150.421} C_VEL
LIN {X 0,Y 664.729,Z 1057.781,A -85,B 0,C 180,E1 5156.043,E2 5156.043} C_VEL
LIN {X 0,Y 669.276,Z 996.027,A -85,B 0,C 180,E1 5160.739,E2 5160.739} C_VEL
LIN {X 0,Y 673.7,Z 928.394,A -85,B 0,C 180,E1 5164.168,E2 5164.168} C_VEL
LIN {X 0,Y 676.976,Z 857.083,A -85,B 0,C 180,E1 5166.323,E2 5166.323} C_VEL
LIN {X 0,Y 676.057,Z 795.62,A -85,B 0,C 180,E1 5167.376,E2 5167.376} C_VEL
LIN {X 0,Y 658.122,Z 762.06,A -85,B 0,C 180,E1 5169.145,E2 5169.145} C_VEL
LIN {X 0,Y 658.241,Z 762.06,A -85,B 0,C 180,E1 5177.157,E2 5177.157} C_VEL
LIN {X 0,Y 658.19,Z 762.06,A -85,B 0,C 180,E1 5185.616,E2 5185.616} C_VEL
LIN {X 0,Y 658.271,Z 762.06,A -85,B 0,C 180,E1 5193.296,E2 5193.296} C_VEL
LIN {X 0,Y 658.379,Z 762.06,A -85,B 0,C 180,E1 5200.486,E2 5200.486} C_VEL
LIN {X 0,Y 659.39,Z 762.06,A -85,B 0,C 180,E1 5208.731,E2 5208.731} C_VEL
LIN {X 0,Y 659.17,Z 762.06,A -85,B 0,C 180,E1 5218.034,E2 5218.034} C_VEL
LIN {X 0,Y 658.911,Z 762.06,A -85,B 0,C 180,E1 5225.963,E2 5225.963} C_VEL
LIN {X 0,Y 658.645,Z 762.06,A -85,B 0,C 180,E1 5234.017,E2 5234.017} C_VEL
LIN {X 0,Y 658.29,Z 762.06,A -85,B 0,C 180,E1 5242.375,E2 5242.375} C_VEL
LIN {X 0,Y 658.343,Z 762.06,A -85,B 0,C 180,E1 5250.249,E2 5250.249} C_VEL
LIN {X 0,Y 658.024,Z 762.06,A -85,B 0,C 180,E1 5253.066,E2 5253.066} C_VEL
LIN {X 0,Y 650.254,Z 762.06,A -85,B 0,C 180,E1 5256.107,E2 5256.107} C_VEL
LIN {X 0,Y 650.337,Z 762.751,A -85,B 0,C 180,E1 5265.952,E2 5265.952} C_VEL
LIN {X 0,Y 675.275,Z 810.756,A -85,B 0,C 180,E1 5268.634,E2 5268.634} C_VEL
LIN {X 0,Y 672.822,Z 889.18,A -85,B 0,C 180,E1 5270.247,E2 5270.247} C_VEL
LIN {X 0,Y 668.084,Z 961.002,A -85,B 0,C 180,E1 5273.018,E2 5273.018} C_VEL
LIN {X 0,Y 662.395,Z 1030.243,A -85,B 0,C 180,E1 5277.161,E2 5277.161} C_VEL
LIN {X 0,Y 657.065,Z 1092.287,A -85,B 0,C 180,E1 5282.544,E2 5282.544} C_VEL
LIN {X 0,Y 653.362,Z 1141.27,A -85,B 0,C 180,E1 5288.58,E2 5288.58} C_VEL
LIN {X 0,Y 651.616,Z 1174.66,A -85,B 0,C 180,E1 5294.475,E2 5294.475} C_VEL
LIN {X 0,Y 650.982,Z 1195.32,A -85,B 0,C 180,E1 5299.936,E2 5299.936} C_VEL
LIN {X 0,Y 650.887,Z 1206.816,A -85,B 0,C 180,E1 5305.321,E2 5305.321} C_VEL
LIN {X 0,Y 651.008,Z 1209.838,A -85,B 0,C 180,E1 5310.666,E2 5310.666} C_VEL
LIN {X 0,Y 651.001,Z 1203.526,A -85,B 0,C 180,E1 5316.687,E2 5316.687} C_VEL
LIN {X 0,Y 651.276,Z 1186.209,A -85,B 0,C 180,E1 5322.779,E2 5322.779} C_VEL
LIN {X 0,Y 652.482,Z 1156.814,A -85,B 0,C 180,E1 5328.944,E2 5328.944} C_VEL
LIN {X 0,Y 655.4,Z 1114.466,A -85,B 0,C 180,E1 5334.977,E2 5334.977} C_VEL
LIN {X 0,Y 659.979,Z 1058.248,A -85,B 0,C 180,E1 5340.646,E2 5340.646} C_VEL
LIN {X 0,Y 665.669,Z 991.973,A -85,B 0,C 180,E1 5345.332,E2 5345.332} C_VEL
LIN {X 0,Y 670.917,Z 921.476,A -85,B 0,C 180,E1 5348.674,E2 5348.674} C_VEL
LIN {X 0,Y 674.574,Z 846.102,A -85,B 0,C 180,E1 5350.8,E2 5350.8} C_VEL
LIN {X 0,Y 674.053,Z 804.114,A -85,B 0,C 180,E1 5351.55,E2 5351.55} C_VEL
LIN {X 0,Y 650.319,Z 762.06,A -85,B 0,C 180,E1 5354.264,E2 5354.264} C_VEL
LIN {X 0,Y 650.596,Z 762.06,A -85,B 0,C 180,E1 5363.529,E2 5363.529} C_VEL
LIN {X 0,Y 650.505,Z 762.06,A -85,B 0,C 180,E1 5371.409,E2 5371.409} C_VEL
LIN {X 0,Y 650.582,Z 762.06,A -85,B 0,C 180,E1 5380.741,E2 5380.741} C_VEL
LIN {X 0,Y 650.952,Z 762.06,A -85,B 0,C 180,E1 5389.915,E2 5389.915} C_VEL
LIN {X 0,Y 651.15,Z 762.06,A -85,B 0,C 180,E1 5397.983,E2 5397.983} C_VEL
LIN {X 0,Y 650.901,Z 762.06,A -85,B 0,C 180,E1 5406.01,E2 5406.01} C_VEL
LIN {X 0,Y 650.426,Z 762.06,A -85,B 0,C 180,E1 5414.63,E2 5414.63} C_VEL
LIN {X 0,Y 650.12,Z 762.06,A -85,B 0,C 180,E1 5422.871,E2 5422.871} C_VEL
LIN {X 0,Y 650.595,Z 762.06,A -85,B 0,C 180,E1 5431.704,E2 5431.704} C_VEL
LIN {X 0,Y 650.365,Z 762.06,A -85,B 0,C 180,E1 5439.907,E2 5439.907} C_VEL
LIN {X 0,Y 650.317,Z 762.06,A -85,B 0,C 180,E1 5448.35,E2 5448.35} C_VEL
LIN {X 0,Y 650.751,Z 763.746,A -85,B 0,C 180,E1 5450.261,E2 5450.261} C_VEL
LIN {X 0,Y 671.116,Z 804.788,A -85,B 0,C 180,E1 5452.332,E2 5452.332} C_VEL
LIN {X 0,Y 669.342,Z 883.385,A -85,B 0,C 180,E1 5453.824,E2 5453.824} C_VEL
LIN {X 0,Y 665.264,Z 952.956,A -85,B 0,C 180,E1 5456.429,E2 5456.429} C_VEL
LIN {X 0,Y 660.256,Z 1019.745,A -85,B 0,C 180,E1 5460.409,E2 5460.409} C_VEL
LIN {X 0,Y 655.894,Z 1076.68,A -85,B 0,C 180,E1 5465.408,E2 5465.408} C_VEL
LIN {X 0,Y 652.842,Z 1122.284,A -85,B 0,C 180,E1 5471.199,E2 5471.199} C_VEL
LIN {X 0,Y 651.341,Z 1152.662,A -85,B 0,C 180,E1 5476.88,E2 5476.88} C_VEL
LIN {X 0,Y 650.954,Z 1171.455,A -85,B 0,C 180,E1 5482.64,E2 5482.64} C_VEL
LIN {X 0,Y 650.771,Z 1179.339,A -85,B 0,C 180,E1 5487.998,E2 5487.998} C_VEL
LIN {X 0,Y 650.997,Z 1178.175,A -85,B 0,C 180,E1 5493.34,E2 5493.34} C_VEL
LIN {X 0,Y 651.125,Z 1167.782,A -85,B 0,C 180,E1 5498.709,E2 5498.709} C_VEL
LIN {X 0,Y 651.782,Z 1145.805,A -85,B 0,C 180,E1 5504.538,E2 5504.538} C_VEL
LIN {X 0,Y 653.687,Z 1109.372,A -85,B 0,C 180,E1 5510.586,E2 5510.586} C_VEL
LIN {X 0,Y 657.157,Z 1059.445,A -85,B 0,C 180,E1 5516.207,E2 5516.207} C_VEL
LIN {X 0,Y 662.096,Z 997.293,A -85,B 0,C 180,E1 5521.023,E2 5521.023} C_VEL
LIN {X 0,Y 666.797,Z 931.029,A -85,B 0,C 180,E1 5524.451,E2 5524.451} C_VEL
LIN {X 0,Y 670.342,Z 861.079,A -85,B 0,C 180,E1 5526.64,E2 5526.64} C_VEL
LIN {X 0,Y 669.912,Z 799.066,A -85,B 0,C 180,E1 5527.734,E2 5527.734} C_VEL
LIN {X 0,Y 649.982,Z 762.06,A -85,B 0,C 180,E1 5529.914,E2 5529.914} C_VEL
LIN {X 0,Y 650.22,Z 762.06,A -85,B 0,C 180,E1 5537.282,E2 5537.282} C_VEL
LIN {X 0,Y 650.237,Z 762.06,A -85,B 0,C 180,E1 5545.135,E2 5545.135} C_VEL
LIN {X 0,Y 650.298,Z 762.06,A -85,B 0,C 180,E1 5552.942,E2 5552.942} C_VEL
LIN {X 0,Y 650.356,Z 762.06,A -85,B 0,C 180,E1 5560.806,E2 5560.806} C_VEL
LIN {X 0,Y 651.383,Z 762.06,A -85,B 0,C 180,E1 5568.59,E2 5568.59} C_VEL
LIN {X 0,Y 651.173,Z 762.06,A -85,B 0,C 180,E1 5578.01,E2 5578.01} C_VEL
LIN {X 0,Y 650.867,Z 762.06,A -85,B 0,C 180,E1 5586.037,E2 5586.037} C_VEL
LIN {X 0,Y 650.426,Z 762.06,A -85,B 0,C 180,E1 5594.619,E2 5594.619} C_VEL
LIN {X 0,Y 650.171,Z 762.06,A -85,B 0,C 180,E1 5602.875,E2 5602.875} C_VEL
LIN {X 0,Y 650.389,Z 762.06,A -85,B 0,C 180,E1 5610.131,E2 5610.131} C_VEL
LIN {X 0,Y 650.254,Z 762.06,A -85,B 0,C 180,E1 5616.107,E2 5616.107} C_VEL
LIN {X 0,Y 641.889,Z 762.06,A -85,B 0,C 180,E1 5619.171,E2 5619.171} C_VEL
LIN {X 0,Y 642.457,Z 763.545,A -85,B 0,C 180,E1 5625.281,E2 5625.281} C_VEL
LIN {X 0,Y 669.247,Z 813.68,A -85,B 0,C 180,E1 5628.22,E2 5628.22} C_VEL
LIN {X 0,Y 666.452,Z 891.661,A -85,B 0,C 180,E1 5629.871,E2 5629.871} C_VEL
LIN {X 0,Y 661.242,Z 964.574,A -85,B 0,C 180,E1 5632.765,E2 5632.765} C_VEL
LIN {X 0,Y 655.037,Z 1033.971,A -85,B 0,C 180,E1 5637.038,E2 5637.038} C_VEL
LIN {X 0,Y 649.347,Z 1095.404,A -85,B 0,C 180,E1 5642.526,E2 5642.526} C_VEL
LIN {X 0,Y 645.488,Z 1143.511,A -85,B 0,C 180,E1 5648.643,E2 5648.643} C_VEL
LIN {X 0,Y 643.643,Z 1176.358,A -85,B 0,C 180,E1 5654.659,E2 5654.659} C_VEL
LIN {X 0,Y 642.982,Z 1197.235,A -85,B 0,C 180,E1 5660.496,E2 5660.496} C_VEL
LIN {X 0,Y 642.918,Z 1206.813,A -85,B 0,C 180,E1 5665.263,E2 5665.263} C_VEL
LIN {X 0,Y 643.023,Z 1209.838,A -85,B 0,C 180,E1 5670.674,E2 5670.674} C_VEL
LIN {X 0,Y 643.003,Z 1203.526,A -85,B 0,C 180,E1 5676.771,E2 5676.771} C_VEL
LIN {X 0,Y 643.308,Z 1186.208,A -85,B 0,C 180,E1 5682.94,E2 5682.94} C_VEL
LIN {X 0,Y 644.626,Z 1157.116,A -85,B 0,C 180,E1 5689.13,E2 5689.13} C_VEL
LIN {X 0,Y 647.759,Z 1114.958,A -85,B 0,C 180,E1 5695.231,E2 5695.231} C_VEL
LIN {X 0,Y 652.784,Z 1058.485,A -85,B 0,C 180,E1 5700.999,E2 5700.999} C_VEL
LIN {X 0,Y 658.949,Z 991.508,A -85,B 0,C 180,E1 5705.778,E2 5705.778} C_VEL
LIN {X 0,Y 664.549,Z 921.473,A -85,B 0,C 180,E1 5709.114,E2 5709.114} C_VEL
LIN {X 0,Y 668.463,Z 846.975,A -85,B 0,C 180,E1 5711.234,E2 5711.234} C_VEL
LIN {X 0,Y 667.913,Z 807.152,A -85,B 0,C 180,E1 5711.975,E2 5711.975} C_VEL
LIN {X 0,Y 642.187,Z 762.06,A -85,B 0,C 180,E1 5714.934,E2 5714.934} C_VEL
LIN {X 0,Y 642.522,Z 762.06,A -85,B 0,C 180,E1 5722.942,E2 5722.942} C_VEL
LIN {X 0,Y 642.476,Z 762.06,A -85,B 0,C 180,E1 5731.018,E2 5731.018} C_VEL
LIN {X 0,Y 642.399,Z 762.06,A -85,B 0,C 180,E1 5739.95,E2 5739.95} C_VEL
LIN {X 0,Y 642.774,Z 762.06,A -85,B 0,C 180,E1 5748.407,E2 5748.407} C_VEL
LIN {X 0,Y 643.174,Z 762.06,A -85,B 0,C 180,E1 5757.958,E2 5757.958} C_VEL
LIN {X 0,Y 642.876,Z 762.06,A -85,B 0,C 180,E1 5766.085,E2 5766.085} C_VEL
LIN {X 0,Y 642.53,Z 762.06,A -85,B 0,C 180,E1 5774.347,E2 5774.347} C_VEL
LIN {X 0,Y 642.12,Z 762.06,A -85,B 0,C 180,E1 5782.94,E2 5782.94} C_VEL
LIN {X 0,Y 642.607,Z 762.06,A -85,B 0,C 180,E1 5790.531,E2 5790.531} C_VEL
LIN {X 0,Y 642.366,Z 762.06,A -85,B 0,C 180,E1 5798.749,E2 5798.749} C_VEL
LIN {X 0,Y 642.111,Z 762.06,A -85,B 0,C 180,E1 5806.113,E2 5806.113} C_VEL
LIN {X 0,Y 642.695,Z 763.838,A -85,B 0,C 180,E1 5809.577,E2 5809.577} C_VEL
LIN {X 0,Y 664.786,Z 807.597,A -85,B 0,C 180,E1 5811.948,E2 5811.948} C_VEL
LIN {X 0,Y 662.76,Z 884.889,A -85,B 0,C 180,E1 5813.455,E2 5813.455} C_VEL
LIN {X 0,Y 658.367,Z 954.291,A -85,B 0,C 180,E1 5816.1,E2 5816.1} C_VEL
LIN {X 0,Y 652.957,Z 1021.175,A -85,B 0,C 180,E1 5820.155,E2 5820.155} C_VEL
LIN {X 0,Y 648.211,Z 1078.291,A -85,B 0,C 180,E1 5825.281,E2 5825.281} C_VEL
LIN {X 0,Y 644.973,Z 1123.383,A -85,B 0,C 180,E1 5831.139,E2 5831.139} C_VEL
LIN {X 0,Y 643.33,Z 1154.063,A -85,B 0,C 180,E1 5837.061,E2 5837.061} C_VEL
LIN {X 0,Y 642.979,Z 1171.454,A -85,B 0,C 180,E1 5842.548,E2 5842.548} C_VEL
LIN {X 0,Y 642.791,Z 1179.339,A -85,B 0,C 180,E1 5847.973,E2 5847.973} C_VEL
LIN {X 0,Y 643.003,Z 1178.176,A -85,B 0,C 180,E1 5853.382,E2 5853.382} C_VEL
LIN {X 0,Y 643.107,Z 1167.784,A -85,B 0,C 180,E1 5858.818,E2 5858.818} C_VEL
LIN {X 0,Y 643.809,Z 1144.805,A -85,B 0,C 180,E1 5864.924,E2 5864.924} C_VEL
LIN {X 0,Y 645.962,Z 1108.364,A -85,B 0,C 180,E1 5870.98,E2 5870.98} C_VEL
LIN {X 0,Y 649.851,Z 1057.361,A -85,B 0,C 180,E1 5876.728,E2 5876.728} C_VEL
LIN {X 0,Y 655.175,Z 995.271,A -85,B 0,C 180,E1 5881.529,E2 5881.529} C_VEL
LIN {X 0,Y 660.311,Z 927.749,A -85,B 0,C 180,E1 5884.992,E2 5884.992} C_VEL
LIN {X 0,Y 664.143,Z 857.174,A -85,B 0,C 180,E1 5887.14,E2 5887.14} C_VEL
LIN {X 0,Y 663.584,Z 801.994,A -85,B 0,C 180,E1 5888.119,E2 5888.119} C_VEL
LIN {X 0,Y 641.929,Z 762.06,A -85,B 0,C 180,E1 5890.518,E2 5890.518} C_VEL
LIN {X 0,Y 642.163,Z 762.06,A -85,B 0,C 180,E1 5898.066,E2 5898.066} C_VEL
LIN {X 0,Y 642.16,Z 762.06,A -85,B 0,C 180,E1 5906.275,E2 5906.275} C_VEL
LIN {X 0,Y 642.275,Z 762.06,A -85,B 0,C 180,E1 5914.091,E2 5914.091} C_VEL
LIN {X 0,Y 642.325,Z 762.06,A -85,B 0,C 180,E1 5921.412,E2 5921.412} C_VEL
LIN {X 0,Y 643.36,Z 762.06,A -85,B 0,C 180,E1 5928.446,E2 5928.446} C_VEL
LIN {X 0,Y 643.197,Z 762.06,A -85,B 0,C 180,E1 5937.985,E2 5937.985} C_VEL
LIN {X 0,Y 642.847,Z 762.06,A -85,B 0,C 180,E1 5946.113,E2 5946.113} C_VEL
LIN {X 0,Y 642.529,Z 762.06,A -85,B 0,C 180,E1 5954.376,E2 5954.376} C_VEL
LIN {X 0,Y 642.147,Z 762.06,A -85,B 0,C 180,E1 5962.97,E2 5962.97} C_VEL
LIN {X 0,Y 642.288,Z 762.06,A -85,B 0,C 180,E1 5970.551,E2 5970.551} C_VEL
LIN {X 0,Y 641.889,Z 762.06,A -85,B 0,C 180,E1 5979.171,E2 5979.171} C_VEL
LIN {X 0,Y 633.811,Z 762.06,A -85,B 0,C 180,E1 5982.285,E2 5982.285} C_VEL
LIN {X 0,Y 634.416,Z 763.542,A -85,B 0,C 180,E1 5984.641,E2 5984.641} C_VEL
LIN {X 0,Y 663.262,Z 815.315,A -85,B 0,C 180,E1 5987.779,E2 5987.779} C_VEL
LIN {X 0,Y 660.205,Z 893.174,A -85,B 0,C 180,E1 5989.463,E2 5989.463} C_VEL
LIN {X 0,Y 654.57,Z 966.273,A -85,B 0,C 180,E1 5992.414,E2 5992.414} C_VEL
LIN {X 0,Y 647.903,Z 1035.443,A -85,B 0,C 180,E1 5996.745,E2 5996.745} C_VEL
LIN {X 0,Y 641.943,Z 1095.458,A -85,B 0,C 180,E1 6002.187,E2 6002.187} C_VEL
LIN {X 0,Y 637.701,Z 1143.509,A -85,B 0,C 180,E1 6008.369,E2 6008.369} C_VEL
LIN {X 0,Y 635.733,Z 1176.119,A -85,B 0,C 180,E1 6014.409,E2 6014.409} C_VEL
LIN {X 0,Y 634.99,Z 1197.235,A -85,B 0,C 180,E1 6020.375,E2 6020.375} C_VEL
LIN {X 0,Y 634.937,Z 1206.81,A -85,B 0,C 180,E1 6025.203,E2 6025.203} C_VEL
LIN {X 0,Y 635.018,Z 1209.838,A -85,B 0,C 180,E1 6030.683,E2 6030.683} C_VEL
LIN {X 0,Y 634.95,Z 1203.015,A -85,B 0,C 180,E1 6037.128,E2 6037.128} C_VEL
LIN {X 0,Y 635.341,Z 1186.207,A -85,B 0,C 180,E1 6043.105,E2 6043.105} C_VEL
LIN {X 0,Y 636.731,Z 1157.98,A -85,B 0,C 180,E1 6049.219,E2 6049.219} C_VEL
LIN {X 0,Y 640.117,Z 1115.729,A -85,B 0,C 180,E1 6055.455,E2 6055.455} C_VEL
LIN {X 0,Y 645.616,Z 1058.313,A -85,B 0,C 180,E1 6061.398,E2 6061.398} C_VEL
LIN {X 0,Y 652.079,Z 993.031,A -85,B 0,C 180,E1 6066.112,E2 6066.112} C_VEL
LIN {X 0,Y 658.121,Z 923.127,A -85,B 0,C 180,E1 6069.498,E2 6069.498} C_VEL
LIN {X 0,Y 662.376,Z 848.396,A -85,B 0,C 180,E1 6071.665,E2 6071.665} C_VEL
LIN {X 0,Y 661.873,Z 810.287,A -85,B 0,C 180,E1 6072.402,E2 6072.402} C_VEL
LIN {X 0,Y 634.109,Z 762.06,A -85,B 0,C 180,E1 6075.579,E2 6075.579} C_VEL
LIN {X 0,Y 634.514,Z 762.06,A -85,B 0,C 180,E1 6084.105,E2 6084.105} C_VEL
LIN {X 0,Y 634.541,Z 762.06,A -85,B 0,C 180,E1 6092.181,E2 6092.181} C_VEL
LIN {X 0,Y 634.619,Z 762.06,A -85,B 0,C 180,E1 6101.148,E2 6101.148} C_VEL
LIN {X 0,Y 634.723,Z 762.06,A -85,B 0,C 180,E1 6111.044,E2 6111.044} C_VEL
LIN {X 0,Y 635.175,Z 762.06,A -85,B 0,C 180,E1 6117.932,E2 6117.932} C_VEL
LIN {X 0,Y 634.834,Z 762.06,A -85,B 0,C 180,E1 6126.162,E2 6126.162} C_VEL
LIN {X 0,Y 634.473,Z 762.06,A -85,B 0,C 180,E1 6134.533,E2 6134.533} C_VEL
LIN {X 0,Y 634.138,Z 762.06,A -85,B 0,C 180,E1 6142.973,E2 6142.973} C_VEL
LIN {X 0,Y 634.58,Z 762.06,A -85,B 0,C 180,E1 6150.93,E2 6150.93} C_VEL
LIN {X 0,Y 634.356,Z 762.06,A -85,B 0,C 180,E1 6159.332,E2 6159.332} C_VEL
LIN {X 0,Y 634.313,Z 762.06,A -85,B 0,C 180,E1 6168.535,E2 6168.535} C_VEL
LIN {X 0,Y 635.61,Z 766.357,A -85,B 0,C 180,E1 6168.997,E2 6168.997} C_VEL
LIN {X 0,Y 658.316,Z 808.091,A -85,B 0,C 180,E1 6171.513,E2 6171.513} C_VEL
LIN {X 0,Y 656.252,Z 885.594,A -85,B 0,C 180,E1 6173.055,E2 6173.055} C_VEL
LIN {X 0,Y 651.527,Z 955.035,A -85,B 0,C 180,E1 6175.735,E2 6175.735} C_VEL
LIN {X 0,Y 645.736,Z 1022.047,A -85,B 0,C 180,E1 6179.855,E2 6179.855} C_VEL
LIN {X 0,Y 640.52,Z 1079.902,A -85,B 0,C 180,E1 6185.151,E2 6185.151} C_VEL
LIN {X 0,Y 637.119,Z 1123.713,A -85,B 0,C 180,E1 6190.952,E2 6190.952} C_VEL
LIN {X 0,Y 635.384,Z 1154.062,A -85,B 0,C 180,E1 6196.896,E2 6196.896} C_VEL
LIN {X 0,Y 634.995,Z 1171.827,A -85,B 0,C 180,E1 6202.619,E2 6202.619} C_VEL
LIN {X 0,Y 634.796,Z 1179.339,A -85,B 0,C 180,E1 6207.948,E2 6207.948} C_VEL
LIN {X 0,Y 634.996,Z 1178.177,A -85,B 0,C 180,E1 6213.424,E2 6213.424} C_VEL
LIN {X 0,Y 635.112,Z 1167.785,A -85,B 0,C 180,E1 6218.93,E2 6218.93} C_VEL
LIN {X 0,Y 635.88,Z 1145.114,A -85,B 0,C 180,E1 6225.051,E2 6225.051} C_VEL
LIN {X 0,Y 638.206,Z 1108.366,A -85,B 0,C 180,E1 6231.247,E2 6231.247} C_VEL
LIN {X 0,Y 642.396,Z 1057.7,A -85,B 0,C 180,E1 6237.03,E2 6237.03} C_VEL
LIN {X 0,Y 648.1,Z 995.613,A -85,B 0,C 180,E1 6241.89,E2 6241.89} C_VEL
LIN {X 0,Y 653.643,Z 928.051,A -85,B 0,C 180,E1 6245.388,E2 6245.388} C_VEL
LIN {X 0,Y 657.74,Z 857.518,A -85,B 0,C 180,E1 6247.555,E2 6247.555} C_VEL
LIN {X 0,Y 657.237,Z 805.084,A -85,B 0,C 180,E1 6248.52,E2 6248.52} C_VEL
LIN {X 0,Y 633.931,Z 762.06,A -85,B 0,C 180,E1 6251.139,E2 6251.139} C_VEL
LIN {X 0,Y 634.107,Z 762.06,A -85,B 0,C 180,E1 6258.883,E2 6258.883} C_VEL
LIN {X 0,Y 634.272,Z 762.06,A -85,B 0,C 180,E1 6267.44,E2 6267.44} C_VEL
LIN {X 0,Y 634.373,Z 762.06,A -85,B 0,C 180,E1 6275.263,E2 6275.263} C_VEL
LIN {X 0,Y 634.757,Z 762.06,A -85,B 0,C 180,E1 6284.054,E2 6284.054} C_VEL
LIN {X 0,Y 634.765,Z 762.06,A -85,B 0,C 180,E1 6291.073,E2 6291.073} C_VEL
LIN {X 0,Y 635.198,Z 762.06,A -85,B 0,C 180,E1 6297.96,E2 6297.96} C_VEL
LIN {X 0,Y 634.805,Z 762.06,A -85,B 0,C 180,E1 6306.191,E2 6306.191} C_VEL
LIN {X 0,Y 634.486,Z 762.06,A -85,B 0,C 180,E1 6314.562,E2 6314.562} C_VEL
LIN {X 0,Y 634.163,Z 762.06,A -85,B 0,C 180,E1 6322.972,E2 6322.972} C_VEL
LIN {X 0,Y 634.171,Z 762.06,A -85,B 0,C 180,E1 6330.985,E2 6330.985} C_VEL
LIN {X 0,Y 633.858,Z 762.06,A -85,B 0,C 180,E1 6339.405,E2 6339.405} C_VEL
LIN {X 0,Y 633.811,Z 762.06,A -85,B 0,C 180,E1 6342.285,E2 6342.285} C_VEL
LIN {X 0,Y 626.116,Z 762.06,A -85,B 0,C 180,E1 6343.678,E2 6343.678} C_VEL
LIN {X 0,Y 629.231,Z 768.597,A -85,B 0,C 180,E1 6344.295,E2 6344.295} C_VEL
LIN {X 0,Y 657.213,Z 820.485,A -85,B 0,C 180,E1 6347.385,E2 6347.385} C_VEL
LIN {X 0,Y 653.683,Z 897.942,A -85,B 0,C 180,E1 6349.15,E2 6349.15} C_VEL
LIN {X 0,Y 647.684,Z 970.453,A -85,B 0,C 180,E1 6352.18,E2 6352.18} C_VEL
LIN {X 0,Y 640.614,Z 1038.528,A -85,B 0,C 180,E1 6356.567,E2 6356.567} C_VEL
LIN {X 0,Y 634.152,Z 1098.787,A -85,B 0,C 180,E1 6362.203,E2 6362.203} C_VEL
LIN {X 0,Y 629.79,Z 1145.88,A -85,B 0,C 180,E1 6368.467,E2 6368.467} C_VEL
LIN {X 0,Y 627.725,Z 1178.865,A -85,B 0,C 180,E1 6374.845,E2 6374.845} C_VEL
LIN {X 0,Y 627.011,Z 1199.023,A -85,B 0,C 180,E1 6380.954,E2 6380.954} C_VEL
LIN {X 0,Y 626.831,Z 1208.374,A -85,B 0,C 180,E1 6386.531,E2 6386.531} C_VEL
LIN {X 0,Y 626.749,Z 1209.405,A -85,B 0,C 180,E1 6392.079,E2 6392.079} C_VEL
LIN {X 0,Y 626.911,Z 1202.167,A -85,B 0,C 180,E1 6397.644,E2 6397.644} C_VEL
LIN {X 0,Y 627.442,Z 1184.867,A -85,B 0,C 180,E1 6403.629,E2 6403.629} C_VEL
LIN {X 0,Y 629.04,Z 1156.008,A -85,B 0,C 180,E1 6409.829,E2 6409.829} C_VEL
LIN {X 0,Y 632.672,Z 1114.136,A -85,B 0,C 180,E1 6415.983,E2 6415.983} C_VEL
LIN {X 0,Y 638.516,Z 1057.655,A -85,B 0,C 180,E1 6421.85,E2 6421.85} C_VEL
LIN {X 0,Y 645.651,Z 990.598,A -85,B 0,C 180,E1 6426.694,E2 6426.694} C_VEL
LIN {X 0,Y 652.036,Z 921.193,A -85,B 0,C 180,E1 6430.026,E2 6430.026} C_VEL
LIN {X 0,Y 656.447,Z 847.63,A -85,B 0,C 180,E1 6432.144,E2 6432.144} C_VEL
LIN {X 0,Y 655.947,Z 813.415,A -85,B 0,C 180,E1 6432.831,E2 6432.831} C_VEL
LIN {X 0,Y 626.06,Z 762.06,A -85,B 0,C 180,E1 6436.275,E2 6436.275} C_VEL
LIN {X 0,Y 626.562,Z 762.06,A -85,B 0,C 180,E1 6445.283,E2 6445.283} C_VEL
LIN {X 0,Y 626.553,Z 762.06,A -85,B 0,C 180,E1 6453.359,E2 6453.359} C_VEL
LIN {X 0,Y 626.553,Z 762.06,A -85,B 0,C 180,E1 6462.947,E2 6462.947} C_VEL
LIN {X 0,Y 626.726,Z 762.06,A -85,B 0,C 180,E1 6470.929,E2 6470.929} C_VEL
LIN {X 0,Y 627.195,Z 762.06,A -85,B 0,C 180,E1 6477.906,E2 6477.906} C_VEL
LIN {X 0,Y 626.802,Z 762.06,A -85,B 0,C 180,E1 6486.242,E2 6486.242} C_VEL
LIN {X 0,Y 626.408,Z 762.06,A -85,B 0,C 180,E1 6494.724,E2 6494.724} C_VEL
LIN {X 0,Y 626.276,Z 762.06,A -85,B 0,C 180,E1 6502.049,E2 6502.049} C_VEL
LIN {X 0,Y 626.55,Z 762.06,A -85,B 0,C 180,E1 6511.371,E2 6511.371} C_VEL
LIN {X 0,Y 626.327,Z 762.06,A -85,B 0,C 180,E1 6520.299,E2 6520.299} C_VEL
LIN {X 0,Y 626.523,Z 764.003,A -85,B 0,C 180,E1 6528.13,E2 6528.13} C_VEL
LIN {X 0,Y 652.214,Z 810.668,A -85,B 0,C 180,E1 6531.069,E2 6531.069} C_VEL
LIN {X 0,Y 649.715,Z 887.27,A -85,B 0,C 180,E1 6532.675,E2 6532.675} C_VEL
LIN {X 0,Y 644.652,Z 956.893,A -85,B 0,C 180,E1 6535.418,E2 6535.418} C_VEL
LIN {X 0,Y 638.441,Z 1023.594,A -85,B 0,C 180,E1 6539.601,E2 6539.601} C_VEL
